// TwinCAT 3 PLC project Lynus_HTTP_Functions
// Title: Lynus HTTP Functions
// Company: Lynus AG
// ProjectVersion: 1.0.0.0
// ProgramVersion: 3.1.4023.0
// libraries:
//   Lynus Standards, * (Lynus AG)
//   Tc2_Standard, * (Beckhoff Automation GmbH)
//   Tc2_System, * (Beckhoff Automation GmbH)
//   Tc2_Utilities, * (Beckhoff Automation GmbH)
//   Tc3_IotBase, * (Beckhoff Automation GmbH)
//   Tc3_JsonXml, * (Beckhoff Automation GmbH)
//   Tc3_Module, * (Beckhoff Automation GmbH)
// project tree:
//   DUTs/Auhofcenter Vienna/ ST_ListOfVariables_Auhofcenter.TcDUT
//   DUTs/SmartMe/ ST_ListOfValues_SmartMe_ElectricMeter.TcDUT
//   DUTs/Suurstoffi Zug/Energy Part/ ST_Values_Energy_Surstoffi.TcDUT
//   DUTs/Suurstoffi Zug/Iosys Part/ ST_Values_Checked_Iosys.TcDUT, ST_Values_Iosys.TcDUT
//   DUTs/Zaptec ECS/ ST_Zaptec_ECS_State.TcDUT, ST_Zaptec_Input_Charger.TcDUT, ST_Zaptec_Input_Installation.TcDUT
//   FBs/Auhofcenter Vienna/Client FBs/ FB_GetSet_Data_Auhofcenter.TcPOU
//   FBs/Auhofcenter Vienna/Helper FBs/ FB_Decode_Json_Auhofcenter.TcPOU, FB_HTTP_Get_Auhofcenter.TcPOU
//   FBs/SmartMe/Client FBs/ FB_Get_Data_SmartMeApi_ElectricMeter.TcPOU
//   FBs/SmartMe/Helper FBs/ FB_Decode_Json_SmartMe_ElectricMeter.TcPOU, FB_HTTP_GetData_Smart_me.TcPOU
//   FBs/Suurstoffi Zug/Energy Part/Client FBs/ FB_Get_Data_Energy_Surstoffi.TcPOU
//   FBs/Suurstoffi Zug/Energy Part/Helper FBs/ FB_Decode_Json_Energy.TcPOU, FB_HTTP_Get_Energy_Surstoffi.TcPOU
//   FBs/Suurstoffi Zug/Iosys Part/Client FBs/ FB_Get_Data_Iosys.TcPOU
//   FBs/Suurstoffi Zug/Iosys Part/Helper FBs/ FB_Check_List_Iosys.TcPOU, FB_Decode_Json_Iosys.TcPOU, FB_HTTP_Get_Iosys.TcPOU
//   FBs/Zaptec ECS/Client FBs/ FB_ECS_HTTP_ZaptecAccount.TcPOU
//   FBs/Zaptec ECS/Helper FBs/ FB_HTTP_Get_Zaptec_ECS_State.TcPOU, FB_HTTP_Post_Zaptec_Current.TcPOU, FB_HTTP_Post_Zaptec_ReqToken.TcPOU

// ---- DUTs/Auhofcenter Vienna/ST_ListOfVariables_Auhofcenter.TcDUT
TYPE ST_ListOfVariables_Auhofcenter :
STRUCT
	bIsString				: BOOL;
	sVariableName			: STRING(15);
	sVariableValue			: STRING(30);
END_STRUCT
END_TYPE

// ---- DUTs/SmartMe/ST_ListOfValues_SmartMe_ElectricMeter.TcDUT
TYPE ST_ListOfValues_SmartMe_ElectricMeter :
STRUCT
	sID					: STRING(50);					//ID from the Device from the Smart-me Project
	sName				: STRING(255);					//Name from the Device from the Smart-me Project
	sActivePowerUnit 	: STRING(20);					//Unit from the Active Power from the Device from the Smart-me Project
	sCounterReadingUnit	: STRING(20);					//Unit from the Counter Reading from the Device from the Smart-me Project
	sValueDate			: STRING(30);					//Date and time when the device last sent data to the Smart Me database
	bNotAllDataIncluded	: BOOL;							//Not all Data from this Structure are included in the Response from the Device from the Smart-me Project  
	bDigitalOutput1		: BOOL;							//State from the Digital Output 1 from the Device from the Smart-me Project 
	bDigitalOutput2		: BOOL;							//State from the Digital Output 2 from the Device from the Smart-me Project
	udiActiveTariff		: UDINT;						//Actual Active tariff from the Device from the Smart-me Project
	uliSerialNr			: ULINT;						//Serial Number from the Device from the Smart-me Project
	lrPowerFactor		: LREAL;						//Power Factor from the Device from the Smart-me Project			
	lrVoltageL1			: LREAL;						//Voltage L1 from the Device from the Smart-me Project	
	lrVoltageL2			: LREAL;						//Voltage L2 from the Device from the Smart-me Project
	lrVoltageL3			: LREAL;						//Voltage L3 from the Device from the Smart-me Project
	lrCurrentL1			: LREAL;						//Current L1 from the Device from the Smart-me Project
	lrCurrentL2			: LREAL;						//Current L2 from the Device from the Smart-me Project
	lrCurrentL3			: LREAL;						//Current L3 from the Device from the Smart-me Project
	lrActivePower		: LREAL;						//Active Power from the Device from the Smart-me Project
	lrActivePowerL1		: LREAL;						//Active Power L1 from the Device from the Smart-me Project
	lrActivePowerL2		: LREAL;						//Active Power L2 from the Device from the Smart-me Project
	lrActivePowerL3		: LREAL;						//Active Power L3 from the Device from the Smart-me Project
	lrCounterReading	: LREAL;						//Counter Reading Value from the Device from the Smart-me Project
	lrCounterReadingT1	: LREAL;						//Counter Reading T1 Value from the Device from the Smart-me Project
	lrCounterReadingT2	: LREAL;						//Counter Reading T2 Value from the Device from the Smart-me Project
	lrCounterReadingT3	: LREAL;						//Counter Reading T3 Value from the Device from the Smart-me Project
	lrCounterReadingT4	: LREAL;						//Counter Reading T4 Value from the Device from the Smart-me Project
	lrCounterReadingImp	: LREAL;						//Counter Reading Import Value from the Device from the Smart-me Project
	lrCounterReadingExp	: LREAL;						//Counter Reading Export Value from the Device from the Smart-me Project
END_STRUCT
END_TYPE

// ---- DUTs/Suurstoffi Zug/Energy Part/ST_Values_Energy_Surstoffi.TcDUT
TYPE ST_Values_Energy_Surstoffi :
STRUCT
	sTimestamp			: STRING(255);						//Timestamp
	sID					: STRING(255);						//Id from the Datapoint
	lrValue				: LREAL;							//Value from the Datapoint
END_STRUCT
END_TYPE

// ---- DUTs/Suurstoffi Zug/Iosys Part/ST_Values_Checked_Iosys.TcDUT
TYPE ST_Values_Checked_Iosys :
STRUCT
	sTimestamp			: STRING(255);						//Timestamp
	sId					: STRING(255);						//Id from the Datapoint
	lrValue				: LREAL;							//Value from Datapoint
END_STRUCT
END_TYPE

// ---- DUTs/Suurstoffi Zug/Iosys Part/ST_Values_Iosys.TcDUT
{attribute 'conditionalshow'}
TYPE ST_Values_Iosys :
STRUCT
	{attribute 'hide'}
	sTimestamp			: STRING(255);					//Timestamp
	{attribute 'hide'}
	sId					: STRING(255);					//Id from the Datapoint
	{attribute 'hide'}
	sValue				: STRING(255);					//Value from Datapoint
	{attribute 'hide'}
	bNoValue			: BOOL;							//Datapoint received but without value
END_STRUCT
END_TYPE

// ---- DUTs/Zaptec ECS/ST_Zaptec_ECS_State.TcDUT
TYPE ST_Zaptec_ECS_State :
STRUCT
	bIsOnline				: BOOL;			//Shows if the Charger is Online
	bIsEnabled				: BOOL;			//Shows if the Charger is Enabled	
	rAllocatedCurrent		: REAL;			//Shows the Allocated Current in A (Only adjustable if you set via the installation API)
	rMaxCurrect				: REAL;			//Max Charge Current from Charging Station in A (Only adjustable if you set via the charger API)
	rMinCurrect				: REAL;			//Min Charge Current from Charging Station in A (Only adjustable if you set via the charger API)
	rCurrentL1				: REAL;			//Current in A from L1
	rCurrentL2				: REAL;			//Current in A from L2
	rCurrentL3				: REAL;			//Current in A from L3
	rPower					: REAL;			//Power in kW
	rEnergySession			: REAL;			//Energy in kWh from the current/last session
	diOperationMode			: DINT;			//Operation Mode form the Charger
	diWarnings				: DINT;			//Warnings from the Charger
	sChargerID				: STRING(50);	//Charger ID from Response
END_STRUCT
END_TYPE

// ---- DUTs/Zaptec ECS/ST_Zaptec_Input_Charger.TcDUT
TYPE ST_Zaptec_Input_Charger :
STRUCT
	rMinCurrentCharger					: REAL;													//Min Current for Charging Station
	rMaxCurrentCharger					: REAL;													//Max Current for Charging Station 
	sChargerID							: STRING(50);											//Charger ID
END_STRUCT
END_TYPE

// ---- DUTs/Zaptec ECS/ST_Zaptec_Input_Installation.TcDUT
TYPE ST_Zaptec_Input_Installation :
STRUCT
	rAvailableCurrentInstallation		: REAL;													//Available Current for Installation
	sInstallationID						: STRING(50);											//Installation ID
END_STRUCT
END_TYPE

// ---- FBs/Auhofcenter Vienna/Client FBs/FB_GetSet_Data_Auhofcenter.TcPOU
{attribute 'hide_all_locals'}
FUNCTION_BLOCK FB_GetSet_Data_Auhofcenter
VAR_INPUT
	bStart						: BOOL;															//Start the connection to the Service
	bWriteRequest				: BOOL;															//Send a Write Request to the Server
	bReadRequest				: BOOL;															//Send a Read Request to the Server
	tDelayRequest				: TIME := T#15S;												//Timer for delay before start with the next read or write Request
	sHostname					: STRING(255);													//Hostname or IP Adress from the Server
	arrListOfVariables			: ARRAY[1..100] OF ST_ListOfVariables_Auhofcenter;				//List of Variables what the function must be send or write		
END_VAR
VAR_OUTPUT
	bValidResult				: BOOL;															//Valid Result received from Server
    bBusy						: BOOL;															//Function is Busy
    bError						: BOOL;															//Error sucess
	bDone						: BOOL;															//True after the decoding from the received Json File
	bConnected					: BOOL;															//Connection to the Server
	arrListOfVariabelsOut		: ARRAY[1..100] OF ST_ListOfVariables_Auhofcenter;				//Received Values form the Server after read or write command
	hrErrorCode       			: HRESULT;														//Error Result from Http Client
END_VAR
VAR
	fbHttpClientEnergyHttp		: FB_IotHttpClient;												//Http Client Function
	fbHttpGet					: FB_HTTP_Get_Auhofcenter;										//Http Get Request to the Server
	fbDecodeJson				: FB_Decode_Json_Auhofcenter;									//Function to decode the received Json File
	timStartRequest				: TON;															//Timer to Start the Request
	timDissableFunctions		: TON;															//Timer to dissable the Function after Lynus_Standards.Constants_General.tTimeDissableLynusFunctions Days without connection to the Lynus Cloud
	timResetConnectionOnGVL		: TON;															//Timer to try reset the connection Flag on the GVL. (When somebody delete the Connection Function and make only a onlinechange)
	timReset24					: TON;															//timer disconnect every 24h
	FPStartRequest				: R_TRIG;														//Internal positive Edge
	FPDone						: R_TRIG;														//Internal positive Edge
	FNStart						: F_TRIG;														//Internal negative Edge
	arrListOfVariablesInt		: ARRAY[1..100] OF ST_ListOfVariables_Auhofcenter;				//Internal List of Variables to compare it with received values after a write Request	
	bErrorCheckValues			: BOOL;															//Error flag to check the values after a write Request
	byLoopCheckValues			: BYTE;															//Loop to check teh values after a Write Request. Server sends the same values back when he has received succesfully
END_VAR

//Creator : Kai Ebensperger
//Company : Lynus AG
//Date : 18.02.2021
//Version : 1.0.0.0

//With this Function is possible to send a HTTP Get Request to the System in the Auhofcenter Vienna
//Its possible to send a Send Request. Here the Server deliver the actual Values.
//On a Write Request we can send new Values to the Server.

(*-------------------------------------------------------------Service from Backend is ready and check the connection to backen for dissabel/enable Function---------------------------------------------------------------*)

//Try to reset the variable for connection on the GVL. When all is normal then the Lynus Mqtt connection function set this variable to true in the next cycle
//When we have no connection to the backend then after Lynus_Standards.Constants_General.tTimeDissableLynusFunctions days the Function is dissabled with all of his functionalities
timResetConnectionOnGVL(IN:= NOT timResetConnectionOnGVL.Q, PT:= T#1H, Q=> , ET=> );
	IF timResetConnectionOnGVL.Q THEN Lynus_Standards.GVL_Communicator.bStateConnectionToEnableFunctions := FALSE; END_IF
		IF NOT Lynus_Standards.GVL_Communicator.bStateConnectionToEnableFunctions THEN timDissableFunctions.IN := TRUE; ELSE timDissableFunctions.IN := FALSE; END_IF  
			timDissableFunctions(IN:= , PT:= Lynus_Standards.Constants_General.tTimeDissableLynusFunctions, Q=> , ET=> );

(*------------------------------------------------------------------------------------Configure HTTP Client------------------------------------------------------------------------------------------------------*)

fbHttpClientEnergyHttp.sHostName := sHostname;
fbHttpClientEnergyHttp.tConnectionTimeout := tDelayRequest;

IF NOT fbHttpClientEnergyHttp.bConfigured THEN 
	fbHttpClientEnergyHttp.nHostPort:= 80;
	fbHttpClientEnergyHttp.stTLS.bNoServerCertCheck:= FALSE;
	fbHttpClientEnergyHttp.bKeepAlive := TRUE;
	fbHttpClientEnergyHttp.tConnectionTimeout := T#10S;
END_IF

//Timer Disconnect to Server every 24H because somthing goes wrog with the loval http plc in the auhofcenter 
timReset24(IN:= bStart AND NOT timReset24.Q, PT:= T#24H, Q=> , ET=> );		

//Timer to start the Request
FPStartRequest(CLK:= bStart, Q=> );
	timStartRequest(IN:= fbHttpClientEnergyHttp.bConfigured AND bStart AND NOT timStartRequest.Q AND NOT timDissableFunctions.Q AND NOT timReset24.Q, PT:= tDelayRequest, Q=> , ET=> );
		IF ((timStartRequest.Q AND NOT bBusy) OR (FPStartRequest.Q AND NOT bBusy AND fbHttpClientEnergyHttp.bConfigured)) THEN fbHttpGet.bSend := TRUE; END_IF

IF timReset24.Q THEN fbHttpGet.bSend := FALSE; END_IF			
		
//Http Get Function
fbHttpGet(
	bWriteRequest:= bWriteRequest, 
	bReadRequest:= bReadRequest, 
	arrListOfVariables:= arrListOfVariables, 
	bSend:= , 
	tTimeOut:= T#20S,
	fbClient:= fbHttpClientEnergyHttp, 
	bValidResult=> bValidResult, 
	bBusy=> bBusy, 
	bError=> ,
	byTypeOfLastRequest=> , 
	sContent=> );

//Copy the values form the actual Request in a internal Array to compare it with the received Values when the request was a Write Request
IF fbHttpGet.bSend THEN arrListOfVariablesInt := arrListOfVariables; END_IF  
	
fbHttpGet.bSend := FALSE;
	
fbDecodeJson(
	bExecute:= fbHttpGet.bValidResult, 
	sContent:= fbHttpGet.sContent, 
	arrListOfVariabels=> arrListOfVariabelsOut, 
	bDone=> bDone, 
	bError=> );

FPDone(CLK:= bDone, Q=> );	
	
//Check after a write command if the Server has received the Values
IF fbHttpGet.byTypeOfLastRequest = 1 AND FPDone.Q THEN
	bErrorCheckValues := FALSE;
		FOR byLoopCheckValues := 1 TO 100 BY 1 DO
			IF arrListOfVariablesInt[byLoopCheckValues].sVariableName <> arrListOfVariabelsOut[byLoopCheckValues].sVariableName OR
				arrListOfVariablesInt[byLoopCheckValues].sVariableValue <> arrListOfVariabelsOut[byLoopCheckValues].sVariableValue THEN
					bErrorCheckValues := TRUE;
			END_IF	 	
		END_FOR 	
END_IF  
	
//Http Client
FNStart(CLK:= bStart, Q=> );
	IF FNStart.Q OR timReset24.Q THEN fbHttpClientEnergyHttp.Disconnect(); END_IF

fbHttpClientEnergyHttp.Execute();

//Connected
bConnected := fbHttpClientEnergyHttp.bConnected;

//Error
IF fbHttpGet.bError OR fbDecodeJson.bError OR fbHttpClientEnergyHttp.bError OR bErrorCheckValues THEN bError := TRUE; ELSE bError := FALSE; END_IF	
	hrErrorCode := fbHttpClientEnergyHttp.hrErrorCode;

END_FUNCTION_BLOCK

// ---- FBs/Auhofcenter Vienna/Helper FBs/FB_HTTP_Get_Auhofcenter.TcPOU
{attribute 'hide_all_locals'}
{attribute 'conditionalshow'}
FUNCTION_BLOCK FB_HTTP_Get_Auhofcenter
VAR_INPUT
	{attribute 'hide'}
	bWriteRequest				: BOOL;													//Send a Write Request to the Server
	{attribute 'hide'}
	bReadRequest				: BOOL;													//Send a Read Request to the Server
	{attribute 'hide'}
	arrListOfVariables			: ARRAY[1..100] OF ST_ListOfVariables_Auhofcenter;		//List of Variables what the function must be send or write
	{attribute 'hide'}
	bSend           			: BOOL;													//Send the Request
	{attribute 'hide'}
	tTimeOut					: TIME := T#10S;										//Timer for Timeout
END_VAR
VAR_IN_OUT
	{attribute 'hide'}
    fbClient          			: FB_IotHttpClient;										//HTTP Client Data
END_VAR
VAR_OUTPUT
	{attribute 'hide'}
	bValidResult				: BOOL;													//Valid Result received from Server
	{attribute 'hide'}
    bBusy             			: BOOL;													//Function is Busy
	{attribute 'hide'}
    bError           			: BOOL;													//Error sucess
	{attribute 'hide'}
	byTypeOfLastRequest			: BYTE;													//Type of the last Request. (0 = Read, 1 = Write)
	{attribute 'hide'}
	sContent         			: STRING(7500);											//Received Content
END_VAR
VAR
    fbRequest        		 	: FB_IotHttpRequest;									//Http Function
	RisingEdge        			: R_TRIG;												//Internal positive edge
	timTimeout					: TON;													//Timer for Timeout
   	bGetContentResult 			: BOOL;													//Get Content Result
	byQuantity					: BYTE;													//Quantity of Datapoints
	byLoop						: BYTE;													//Variable foor Loop to prepear the URI
	nState						: UDINT;												//Statemaschine
  	nReqCount					: UDINT;												//Counter requests
    nResCount					: UDINT;												//Counter results
    nValidResCount				: UDINT;												//Counter valid results
    nErrCount					: UDINT;												//Error Counter
	eErrorCode					: ETcIotHttpRequestError;								//Error Code
	sUriStart					: STRING(20);											//Start URI
	sUriComplete				: STRING(2000);											//Complete URI
END_VAR

//Creator : Kai Ebensperger
//Company : Lynus AG
//Date : 15.07.2021
//Version : 1.0.0.0

//With this Function is possible to send a HTTP Get Request to the System in the Auhof Center in Vienna.

//Timer for Timeout
timTimeout(IN:= nState = 1 AND bBusy, PT:= tTimeOut, Q=> , ET=> );
	IF timTimeout.Q THEN nState := 0; bBusy := FALSE; END_IF

RisingEdge(CLK:= bSend);

CASE nState OF
0:
    IF RisingEdge.Q THEN
		
		byQuantity := 0;
			FOR byLoop := 1 TO 100 BY 1 DO
				IF arrListOfVariables[byLoop].sVariableName <> '' THEN byQuantity := byQuantity + 1; END_IF 
			END_FOR
	
		sUriComplete := '';
			//Read Request
			IF bReadRequest THEN 
				sUriStart := '/lynus/read?';
					sUriComplete := sUriStart;
						IF byQuantity <= 100 THEN
							FOR byLoop := 1 TO byQuantity BY 1 DO
								CONCAT2(ADR(sUriComplete),ADR(arrListOfVariables[byLoop].sVariableName),ADR(sUriComplete),SIZEOF(sUriComplete));
									IF byLoop <= (byQuantity - 1) THEN CONCAT2(ADR(sUriComplete),ADR(','),ADR(sUriComplete),SIZEOF(sUriComplete)); END_IF	
							END_FOR
						END_IF
							byTypeOfLastRequest := 0;
			END_IF
				//Write Request
				IF bWriteRequest THEN 
					sUriStart := '/lynus/write?';
						sUriComplete := sUriStart;
							IF byQuantity <= 100 THEN
								FOR byLoop := 1 TO byQuantity BY 1 DO
									CONCAT2(ADR(sUriComplete),ADR(arrListOfVariables[byLoop].sVariableName),ADR(sUriComplete),SIZEOF(sUriComplete));
										CONCAT2(ADR(sUriComplete),ADR('='),ADR(sUriComplete),SIZEOF(sUriComplete));
											IF arrListOfVariables[byLoop].bIsString THEN CONCAT2(ADR(sUriComplete),ADR('"'),ADR(sUriComplete),SIZEOF(sUriComplete)); END_IF 	
												CONCAT2(ADR(sUriComplete),ADR(arrListOfVariables[byLoop].sVariableValue),ADR(sUriComplete),SIZEOF(sUriComplete));
													IF arrListOfVariables[byLoop].bIsString THEN CONCAT2(ADR(sUriComplete),ADR('"'),ADR(sUriComplete),SIZEOF(sUriComplete)); END_IF 			
														IF byLoop <= (byQuantity - 1) THEN CONCAT2(ADR(sUriComplete),ADR(','),ADR(sUriComplete),SIZEOF(sUriComplete)); END_IF	
								END_FOR
							END_IF
								byTypeOfLastRequest := 1;	
				END_IF
		
		bValidResult := FALSE;
		
		IF fbRequest.SendRequest(sUri:= sUriComplete,
								 fbClient:= fbClient, 
									eRequestType:= ETcIotHttpRequestType.HTTP_Get, 0, 0, 0) THEN
			nState:= 1;
			nReqCount:= nReqCount+1;
			bBusy:= TRUE;
			bError:= FALSE;
		END_IF
    END_IF
	
1:
    IF NOT fbRequest.bBusy THEN
       IF NOT fbRequest.bError THEN
            bGetContentResult:= fbRequest.GetContent(pContent:= ADR(sContent), 
                                                     nContentSize:= SIZEOF(sContent), 
                                                     bSetNullTermination:= TRUE);
            IF fbRequest.nStatusCode >= 200 AND fbRequest.nStatusCode < 300 THEN
                	bValidResult := TRUE;
                    nValidResCount:= nValidResCount+1;
                    bError:= FALSE;
               		nResCount:= nResCount+1;
           END_IF
		   		//Error Response from the Server
				IF sContent = 'Error' THEN bError := TRUE; END_IF
        END_IF
			IF fbRequest.bError THEN bError:= TRUE; eErrorCode := fbRequest.eErrorId; END_IF 
			nState:= 0;
			bBusy:= FALSE;
			IF bError THEN
				nErrCount:= nErrCount+1;
			END_IF	
    END_IF
	
END_CASE

END_FUNCTION_BLOCK

// ---- FBs/Auhofcenter Vienna/Helper FBs/FB_Decode_Json_Auhofcenter.TcPOU
{attribute 'hide_all_locals'}
{attribute 'conditionalshow'}
FUNCTION_BLOCK FB_Decode_Json_Auhofcenter
VAR_INPUT
	{attribute 'hide'}
	bExecute						: BOOL;																			//Start the decoding from the Json File
	{attribute 'hide'}
	sContent         				: STRING(7500);																	//Received Content
END_VAR
VAR_OUTPUT
	{attribute 'hide'}
	arrListOfVariabels				: ARRAY[1..100] OF ST_ListOfVariables_Auhofcenter;								//List with all received Values from the Server
	{attribute 'hide'}
	bDone							: BOOL;																			//True when the decoding is done
	{attribute 'hide'}
	bError							: BOOL;																			//Error Bit
END_VAR
VAR
	fbJsonRead					    : FB_JsonDomParser;																//FB Json Dom reader
 	jsonDocInit  					: SJsonValue;																	//Json value
	jsonDoc		  					: SJsonValue;																	//Json value
	jsonPropID   					: SJsonValue;																	//Json value
	jsonIteratorArrayStart			: SJsonAIterator;																//Json AIterator
	jsonIteratorArrayEnd			: SJsonAIterator;																//Json AIterator
	FPExecute						: R_TRIG;																		//Internal positive edge
	byCounterForArray				: BYTE;																			//Counter to fill the output array with conntent
	byLoopInit						: BYTE;																			//Loop to clear the output array before fill the new content inside
END_VAR

//Creator : Kai Ebensperger
//Company : Lynus AG
//Date : 15.07.2021
//Version : 1.0.0.0

//With this Function we can decode the received Json form the System in the Auhofcenter in Vienna

bDone := FALSE;

FPExecute(CLK:= bExecute, Q=> );

//Start with the Json Doc
jsonDocInit := fbJsonRead.ParseDocument(sContent);

IF FPExecute.Q THEN
	byCounterForArray := 0;	
		bError := FALSE;

	//Clear the Output for new Values
	FOR byLoopInit := 1 TO 100 BY 1 DO
		arrListOfVariabels[byLoopInit].bIsString := FALSE;
			arrListOfVariabels[byLoopInit].sVariableName := '';
				arrListOfVariabels[byLoopInit].sVariableValue := '';
	END_FOR
	
	//Check if the values are inside of a Array 		
	IF jsonDocInit <> 0 THEN
		IF fbJsonRead.IsArray(jsonDocInit) THEN
			jsonIteratorArrayStart := fbJsonRead.ArrayBegin(jsonDocInit);	
				jsonIteratorArrayEnd := fbJsonRead.ArrayEnd(jsonDocInit);
		ELSE
			bError := TRUE;
		END_IF
	ELSE
		bError := TRUE;
	END_IF
		//Start to Decode the Json File
		IF jsonDocInit <> 0 AND jsonIteratorArrayStart <> 0 AND jsonIteratorArrayEnd <> 0 AND NOT bError THEN
		
			WHILE jsonIteratorArrayStart <> jsonIteratorArrayEnd DO  
				jsonDoc := fbJsonRead.GetArrayValue(jsonIteratorArrayStart);
					//Find the Member ID
					jsonPropID := fbJsonRead.FindMember(jsonDoc, 'ID');	
						IF jsonPropID <> 0 THEN
							IF fbJsonRead.IsString(jsonPropID) THEN
								byCounterForArray := byCounterForArray + 1;
									byCounterForArray := LIMIT(1,byCounterForArray,100);	
										arrListOfVariabels[byCounterForArray].sVariableName := fbJsonRead.GetString(jsonPropID);
							ELSE
								bError := TRUE;	
							END_IF	
						END_IF 
					//Find the Member v
					jsonPropID := fbJsonRead.FindMember(jsonDoc, 'v');
						IF jsonPropID <> 0 THEN
							IF fbJsonRead.IsNumber(jsonPropID) THEN
								arrListOfVariabels[byCounterForArray].sVariableValue := LREAL_TO_STRING(fbJsonRead.GetDouble(jsonPropID));
							ELSE
								bError := TRUE;		
							END_IF
						END_IF
					//Find the Member vs
					jsonPropID := fbJsonRead.FindMember(jsonDoc, 'vs');
						IF jsonPropID <> 0 THEN
							IF fbJsonRead.IsString(jsonPropID) THEN
								arrListOfVariabels[byCounterForArray].sVariableValue := fbJsonRead.GetString(jsonPropID);
									arrListOfVariabels[byCounterForArray].bIsString := TRUE;
							ELSE
								bError := TRUE;	
							END_IF
						END_IF
					jsonIteratorArrayStart := fbJsonRead.NextArray(jsonIteratorArrayStart);
			END_WHILE
				bDone := TRUE;
		END_IF
END_IF

END_FUNCTION_BLOCK

// ---- FBs/SmartMe/Client FBs/FB_Get_Data_SmartMeApi_ElectricMeter.TcPOU
{attribute 'hide_all_locals'}
FUNCTION_BLOCK FB_Get_Data_SmartMeApi_ElectricMeter
VAR_INPUT
	bStart						: BOOL;															//Start the connection to the Service
	sUsername					: STRING(50);													//Username from the smart-me Project
	sPassword					: STRING(50);													//Password from the smart-me Project
	tDelayRequest				: TIME := T#1S; 												//Delay between the Requests		
END_VAR
VAR_OUTPUT
	bValidResult				: BOOL;															//Valid Result received from Server
    bBusy						: BOOL;															//Function is Busy
    bError						: BOOL;															//Error sucess
	hrErrorCode       			: HRESULT;														//Error Result from Http Client
	arrListOfDevices			: ARRAY[1..50] OF ST_ListOfValues_SmartMe_ElectricMeter;		//List with all received Values from the Server
END_VAR
VAR
	fbHttpClientSmartMe			: FB_IotHttpClient :=(sHostName:='smart-me.com',
                                  bKeepAlive:=TRUE, tConnectionTimeout:=T#15S);					//Http Client Function
	fbHttpGet					: FB_HTTP_GetData_Smart_me;										//Http Get Request to the Smart Me Service
	fbJson						: FB_Decode_Json_SmartMe_ElectricMeter;							//Deconde received Json
	timStartRequest				: TON;															//Timer to Start the Request
	timDissableFunctions		: TON;															//Timer to dissable the Function after Lynus_Standards.Constants_General.tTimeDissableLynusFunctions Days without connection to the Lynus Cloud
	timResetConnectionOnGVL		: TON;															//Timer to try reset the connection Flag on the GVL. (When somebody delete the Connection Function and make only a onlinechange)
	timReset24					: TON;															//timer disconnect every 24h
	FPStartRequest				: R_TRIG;														//Internal positive Edge
	FNStart						: F_TRIG;														//Internal negative Edge
END_VAR

//Creator : Kai Ebensperger
//Company : Lynus AG
//Date : 29.09.2021
//Version : 1.0.0.0

//With this Function is possible to send a HTTP Get Request to the Smart-me System and recieve values from the Project wich is defined with the Username and the password
//With this Function is possible to decode only Data from Electric Meter in the Project
//Other Device Types or Meters are not supported and the Function deliver a Error
//Attetnion : If the Username is a Mailadress write all in small carakters. For example kai.ebensperger@ventus.ag

(*--------------------------------------------------------------------------------------------------------Limits---------------------------------------------------------------------------------------------------*)

tDelayRequest := LIMIT(T#1S,tDelayRequest,T#15M);

(*-------------------------------------------------------------Service from Backend is ready and check the connection to backen for dissabel/enable Function---------------------------------------------------------------*)

//Try to reset the variable for connection on the GVL. When all is normal then the Lynus Mqtt connection function set this variable to true in the next cycle
//When we have no connection to the backend then after Lynus_Standards.Constants_General.tTimeDissableLynusFunctions days the Function is dissabled with all of his functionalities
timResetConnectionOnGVL(IN:= NOT timResetConnectionOnGVL.Q, PT:= T#1H, Q=> , ET=> );
	IF timResetConnectionOnGVL.Q THEN Lynus_Standards.GVL_Communicator.bStateConnectionToEnableFunctions := FALSE; END_IF
		IF NOT Lynus_Standards.GVL_Communicator.bStateConnectionToEnableFunctions THEN timDissableFunctions.IN := TRUE; ELSE timDissableFunctions.IN := FALSE; END_IF  
			timDissableFunctions(IN:= , PT:= Lynus_Standards.Constants_General.tTimeDissableLynusFunctions, Q=> , ET=> );

(*------------------------------------------------------------------------------------Configure HTTP Client------------------------------------------------------------------------------------------------------*)

IF NOT fbHttpClientSmartMe.bConfigured THEN
    fbHttpClientSmartMe.nHostPort:= 443;
    fbHttpClientSmartMe.stTLS.bNoServerCertCheck:= TRUE;
END_IF

//Timer Disconnect to Server every 24H because somthing goes wrog with the loval http plc in the auhofcenter 
timReset24(IN:= bStart AND NOT timReset24.Q, PT:= T#24H, Q=> , ET=> );

//Timer to start the Request
FPStartRequest(CLK:= bStart, Q=> );
	timStartRequest(IN:= bStart AND NOT timStartRequest.Q AND NOT timDissableFunctions.Q AND NOT bBusy AND fbHttpClientSmartMe.bConfigured AND NOT timReset24.Q, PT:= tDelayRequest, Q=> , ET=> );
		IF timStartRequest.Q OR (FPStartRequest.Q AND NOT bBusy AND fbHttpClientSmartMe.bConfigured) THEN fbHttpGet.bSend := TRUE; END_IF

IF timReset24.Q THEN fbHttpGet.bSend := FALSE; END_IF				
		
//Http Get Function
fbHttpGet(
	bSend:= , 
	sUsername:= sUsername, 
	sPassword:= sPassword, 
	tTimeOut:= T#20S,
	fbClient:= fbHttpClientSmartMe, 
	bValidResult=> bValidResult, 
	bBusy=> bBusy, 
	bError=> , 
	sContent=> );
	
fbHttpGet.bSend := FALSE;
	
//Decode Json
fbJson(
	bExecute:= bValidResult, 
	sContent:= fbHttpGet.sContent, 
	arrListOfDevices=> , 
	bDone=> , 
	bError=> );

IF fbJson.bDone AND NOT fbJson.bError AND NOT bBusy THEN
	arrListOfDevices := fbJson.arrListOfDevices;
END_IF		
	
//Http Client
FNStart(CLK:= bStart, Q=> );
	IF FNStart.Q OR timReset24.Q THEN fbHttpClientSmartMe.Disconnect(); END_IF

fbHttpClientSmartMe.Execute();

//Error
IF fbHttpGet.bError OR fbJson.bError OR fbHttpClientSmartMe.bError THEN bError := TRUE; ELSE bError := FALSE; END_IF	
	hrErrorCode := fbHttpClientSmartMe.hrErrorCode;

END_FUNCTION_BLOCK

// ---- FBs/SmartMe/Helper FBs/FB_HTTP_GetData_Smart_me.TcPOU
{attribute 'hide_all_locals'}
{attribute 'conditionalshow'}
FUNCTION_BLOCK FB_HTTP_GetData_Smart_me
VAR_INPUT
	{attribute 'hide'}
   	bSend               : BOOL;													//Send the Request to the Service
	{attribute 'hide'}
	sUsername			: STRING(50);											//Username from the smart-me Project
	{attribute 'hide'}
	sPassword			: STRING(50);											//Password from the smart-me Project
	{attribute 'hide'}
	tTimeOut			: TIME := T#10S;										//Timer for Timeout
END_VAR
VAR_IN_OUT
	{attribute 'hide'}
    fbClient            : FB_IotHttpClient;										//Connection to the HTTP Client Function
END_VAR
VAR_OUTPUT
	{attribute 'hide'}
	bValidResult		: BOOL;													//Valid Result received from Server
	{attribute 'hide'}
    bBusy               : BOOL;													//Function is Busy
	{attribute 'hide'}
    bError              : BOOL;													//Function has a error
	{attribute 'hide'}
	sContent            : STRING(30000);										//Received Content
END_VAR
VAR
	fbRequest           : FB_IotHttpRequest;									//Http Request Function
    fbHeader            : FB_IotHttpHeaderFieldMap;								//Header Function
	fbJsonWrite     	: FB_JsonSaxWriter;										//Json Write function to generate the based64 Part for the Header
 	timTimeout			: TON;													//Timer for Timeout
	RisingEdge          : R_TRIG;												//Internal rising edge
   	bGetContentResult   : BOOL;													//True when we receive content												
    nState              : UDINT;												//Statemachine for the http request
    nReqCount           : UDINT;												//Request Counter
    nResCount           : UDINT;												//Receive Counter
    nValidResCount      : UDINT;												//Valid Receive Counter
    nErrCount           : UDINT;												//Error Counter
    bOnce               : BOOL:= TRUE;											//Add the addidional Header Part
	sbase64				: STRING(255);											//Based 64 string from the username and Password
	sbase64_CP			: STRING(255);											//Based 64 string from the username and Password to compare it and modify the header
	sCompleteString		: STRING(101);											//Complete string with username and password
	iLen				: INT;													//Lengh from the string
END_VAR

//Creator : Kai Ebensperger
//Company : Lynus AG
//Date : 29.09.2021
//Version : 1.0.0.0

//With this Function its possible to make a Request to the smart-me Database to receive Information from a Project and his devices.

//Convert the Username and the password from string to Ascii and then in a Based64 format
sCompleteString := CONCAT(CONCAT(sUsername,':'),sPassword);
	iLen := LEN(sCompleteString); 
		fbJsonWrite.AddBase64(ADR(sCompleteString),iLen);
			sbase64 := fbJsonWrite.GetDocument();
				fbJsonWrite.ResetDocument();

sbase64 := DELETE(sbase64,1,FIND(sbase64,'"'));	
	sbase64 := DELETE(sbase64,1,FIND(sbase64,'"'));		
	
sbase64 := CONCAT('Basic ',sbase64);

//Add Username and Password to the Header of the Request
IF sbase64 <> sbase64_CP AND nState = 0 THEN bOnce := TRUE; sbase64_CP := sbase64; END_IF  

IF bOnce THEN
    fbHeader.AddField('Authorization',sbase64, FALSE);
    bOnce:= FALSE;
END_IF

//Timer for Timeout
timTimeout(IN:= nState = 1 AND bBusy, PT:= tTimeOut, Q=> , ET=> );
	IF timTimeout.Q THEN nState := 0; bBusy := FALSE; END_IF

//Statemachine to generate the Request

RisingEdge(CLK:= bSend);
	CASE nState OF
		
		0://Request
			IF RisingEdge.Q THEN
				IF fbRequest.SendRequest(sUri:= '/api/Devices', fbClient:= fbClient, 
										 eRequestType:= ETcIotHttpRequestType.HTTP_GET, 0, 0, fbHeader) THEN
					nState:= 1;
					nReqCount:= nReqCount + 1;
					bBusy:= TRUE;
					bError:= FALSE;
					bValidResult := FALSE;
				END_IF
			END_IF
			
		1://Wait for the Response
			IF NOT fbRequest.bBusy THEN
				bError:= TRUE;
					IF NOT fbRequest.bError THEN
						bGetContentResult:= fbRequest.GetContent(pContent:= ADR(sContent),
																 nContentSize:= SIZEOF(sContent), 
																 bSetNullTermination:= TRUE);
						IF fbRequest.nStatusCode >= 200 AND fbRequest.nStatusCode < 300 THEN
							bValidResult := TRUE;
							nResCount:= nResCount + 1;
							bError:= FALSE;
						END_IF
					END_IF
						nState:= 0;
						bBusy:= FALSE;
							IF bError THEN
								nErrCount:= nErrCount + 1;
							END_IF
			END_IF
			
	END_CASE

END_FUNCTION_BLOCK

// ---- FBs/SmartMe/Helper FBs/FB_Decode_Json_SmartMe_ElectricMeter.TcPOU
{attribute 'hide_all_locals'}
{attribute 'conditionalshow'}
FUNCTION_BLOCK FB_Decode_Json_SmartMe_ElectricMeter
VAR_INPUT
	{attribute 'hide'}
	bExecute						: BOOL;																			//Start the decoding from the Json File
	{attribute 'hide'}
	sContent         				: STRING(30000);																//Received Content
END_VAR
VAR_OUTPUT
	{attribute 'hide'}
	arrListOfDevices				: ARRAY[1..50] OF ST_ListOfValues_SmartMe_ElectricMeter;						//List with all received Values from the Server
	{attribute 'hide'}
	bDone							: BOOL;																			//True when the decoding is done
	{attribute 'hide'}
	bError							: BOOL;																			//Error Bit
END_VAR
VAR
	fbJsonRead					    : FB_JsonDomParser;																//FB Json Dom reader
 	jsonDocInit  					: SJsonValue;																	//Json value
	jsonDoc		  					: SJsonValue;																	//Json value
	jsonPropID   					: SJsonValue;																	//Json value
	jsonIteratorArrayStart			: SJsonAIterator;																//Json AIterator
	jsonIteratorArrayEnd			: SJsonAIterator;																//Json AIterator
	FPExecute						: R_TRIG;																		//Internal positive edge
	byCounterForArray				: BYTE;																			//Counter to fill the output array with conntent
	byLoopInit						: BYTE;																			//Loop to clear the output array before fill the new content inside
END_VAR

//Creator : Kai Ebensperger
//Company : Lynus AG
//Date : 29.09.2021
//Version : 1.0.0.0

//With this Function we can decode the received Json form a Smart-Me Project
//With this Function its possible to decode only the Data from Electric Meter from the Smart-me Project
//Other Devices are not supported with this function 

bDone := FALSE;

FPExecute(CLK:= bExecute, Q=> );

//Start with the Json Doc
jsonDocInit := fbJsonRead.ParseDocument(sContent);

IF FPExecute.Q THEN
	byCounterForArray := 0;	
		bError := FALSE;

	//Clear the Output for new Values
	FOR byLoopInit := 1 TO 50 BY 1 DO
		arrListOfDevices[byLoopInit].lrActivePower := 0;
			arrListOfDevices[byLoopInit].sActivePowerUnit := '';
				arrListOfDevices[byLoopInit].sID := '';
					arrListOfDevices[byLoopInit].sName := '';
						arrListOfDevices[byLoopInit].uliSerialNr := 0;
							arrListOfDevices[byLoopInit].sValueDate := '';	
								arrListOfDevices[byLoopInit].sCounterReadingUnit := '';
									arrListOfDevices[byLoopInit].bDigitalOutput1 := FALSE;
										arrListOfDevices[byLoopInit].bDigitalOutput2 := FALSE;
											arrListOfDevices[byLoopInit].bNotAllDataIncluded := FALSE;
												arrListOfDevices[byLoopInit].udiActiveTariff := 0;
													arrListOfDevices[byLoopInit].lrPowerFactor := 0;
														arrListOfDevices[byLoopInit].lrVoltageL1 := 0;
															arrListOfDevices[byLoopInit].lrVoltageL2 := 0;
																arrListOfDevices[byLoopInit].lrVoltageL3 := 0;
																	arrListOfDevices[byLoopInit].lrCurrentL1 := 0;
																		arrListOfDevices[byLoopInit].lrCurrentL2 := 0;
																			arrListOfDevices[byLoopInit].lrCurrentL3 := 0;
																				arrListOfDevices[byLoopInit].lrActivePowerL1 := 0;
																					arrListOfDevices[byLoopInit].lrActivePowerL2 := 0;
																						arrListOfDevices[byLoopInit].lrActivePowerL3 := 0;
																							arrListOfDevices[byLoopInit].lrCounterReading := 0;
																								arrListOfDevices[byLoopInit].lrCounterReadingT1 := 0;
																									arrListOfDevices[byLoopInit].lrCounterReadingT2 := 0;
																										arrListOfDevices[byLoopInit].lrCounterReadingT3 := 0;
																											arrListOfDevices[byLoopInit].lrCounterReadingT4 := 0;
																												arrListOfDevices[byLoopInit].lrCounterReadingImp := 0;	
																													arrListOfDevices[byLoopInit].lrCounterReadingExp := 0;
	END_FOR
	
	//Check if the values are inside of a Array 		
	IF jsonDocInit <> 0 THEN
		IF fbJsonRead.IsArray(jsonDocInit) THEN
			jsonIteratorArrayStart := fbJsonRead.ArrayBegin(jsonDocInit);	
				jsonIteratorArrayEnd := fbJsonRead.ArrayEnd(jsonDocInit);
		ELSE
			bError := TRUE;
		END_IF
	ELSE
		bError := TRUE;
	END_IF
		//Start to Decode the Json File
		IF jsonDocInit <> 0 AND jsonIteratorArrayStart <> 0 AND jsonIteratorArrayEnd <> 0 AND NOT bError THEN
		
			WHILE jsonIteratorArrayStart <> jsonIteratorArrayEnd DO  
				jsonDoc := fbJsonRead.GetArrayValue(jsonIteratorArrayStart);
(*--------------------------------------------------------------------------------------------------Must have Members--------------------------------------------------------------------------------------------------------*)
					//Find the Member Id
					jsonPropID := fbJsonRead.FindMember(jsonDoc, 'Id');	
						IF jsonPropID <> 0 THEN
							IF fbJsonRead.IsString(jsonPropID) THEN
								byCounterForArray := byCounterForArray + 1;
									byCounterForArray := LIMIT(1,byCounterForArray,50);	
										arrListOfDevices[byCounterForArray].sID := fbJsonRead.GetString(jsonPropID);
							ELSE
								bError := TRUE;	
							END_IF	
						END_IF 
					//Find the Member Name
					jsonPropID := fbJsonRead.FindMember(jsonDoc, 'Name');
						IF jsonPropID <> 0 THEN
							IF fbJsonRead.IsString(jsonPropID) THEN
								arrListOfDevices[byCounterForArray].sName := fbJsonRead.GetString(jsonPropID);
							ELSE
								bError := TRUE;		
							END_IF
						END_IF
					//Find the Member Serial
					jsonPropID := fbJsonRead.FindMember(jsonDoc, 'Serial');
						IF jsonPropID <> 0 THEN
							IF fbJsonRead.IsUint64(jsonPropID) THEN
								arrListOfDevices[byCounterForArray].uliSerialNr := fbJsonRead.GetUint64(jsonPropID);
							ELSE
								bError := TRUE;	
							END_IF
						END_IF
					//Find the Member Active Power
					jsonPropID := fbJsonRead.FindMember(jsonDoc, 'ActivePower');
						IF jsonPropID <> 0 THEN
							IF fbJsonRead.IsNumber(jsonPropID) THEN
								arrListOfDevices[byCounterForArray].lrActivePower := fbJsonRead.GetDouble(jsonPropID);
									//Limit for 2 commas
									IF arrListOfDevices[byCounterForArray].lrActivePower >= - 999999999999999 AND arrListOfDevices[byCounterForArray].lrActivePower <= 999999999999999 THEN
										arrListOfDevices[byCounterForArray].lrActivePower := LINT_TO_LREAL(LREAL_TO_LINT((arrListOfDevices[byCounterForArray].lrActivePower) * 100)) / 100;	
									END_IF 
							ELSE
								bError := TRUE;		
							END_IF
						END_IF
					//Find the Member Active Power Unit
					jsonPropID := fbJsonRead.FindMember(jsonDoc, 'ActivePowerUnit');
						IF jsonPropID <> 0 THEN
							IF fbJsonRead.IsString(jsonPropID) THEN
								arrListOfDevices[byCounterForArray].sActivePowerUnit := fbJsonRead.GetString(jsonPropID);
							ELSE
								bError := TRUE;		
							END_IF
						END_IF
					//Find the Member Value Date
					jsonPropID := fbJsonRead.FindMember(jsonDoc, 'ValueDate');
						IF jsonPropID <> 0 THEN
							IF fbJsonRead.IsString(jsonPropID) THEN
								arrListOfDevices[byCounterForArray].sValueDate := fbJsonRead.GetString(jsonPropID);
							ELSE
								bError := TRUE;		
							END_IF
						END_IF
(*--------------------------------------------------------------------------------------------------Additional Members--------------------------------------------------------------------------------------------------------*)
					//Find the Member Counter Reading Unit
					jsonPropID := fbJsonRead.FindMember(jsonDoc, 'CounterReadingUnit');
						IF jsonPropID <> 0 THEN
							IF fbJsonRead.IsString(jsonPropID) THEN
								arrListOfDevices[byCounterForArray].sCounterReadingUnit := fbJsonRead.GetString(jsonPropID);
							END_IF
						ELSE
							arrListOfDevices[byCounterForArray].bNotAllDataIncluded := TRUE;
						END_IF
					//Find the Member Digital Output 1
					jsonPropID := fbJsonRead.FindMember(jsonDoc, 'DigitalOutput1');
						IF jsonPropID <> 0 THEN
							IF fbJsonRead.IsBool(jsonPropID) THEN
								arrListOfDevices[byCounterForArray].bDigitalOutput1 := fbJsonRead.GetBool(jsonPropID);
							END_IF
						ELSE
							arrListOfDevices[byCounterForArray].bNotAllDataIncluded := TRUE;
						END_IF
					//Find the Member Digital Output 2
					jsonPropID := fbJsonRead.FindMember(jsonDoc, 'DigitalOutput2');
						IF jsonPropID <> 0 THEN
							IF fbJsonRead.IsBool(jsonPropID) THEN
								arrListOfDevices[byCounterForArray].bDigitalOutput2 := fbJsonRead.GetBool(jsonPropID);
							END_IF
						ELSE
							arrListOfDevices[byCounterForArray].bNotAllDataIncluded := TRUE;
						END_IF
					//Find the Member ActiveTariff
					jsonPropID := fbJsonRead.FindMember(jsonDoc, 'ActiveTariff');
						IF jsonPropID <> 0 THEN
							IF fbJsonRead.IsUint(jsonPropID) THEN
								arrListOfDevices[byCounterForArray].udiActiveTariff := fbJsonRead.GetUint(jsonPropID);
							END_IF
						ELSE
							arrListOfDevices[byCounterForArray].bNotAllDataIncluded := TRUE;
						END_IF
					//Find the Member PowerFactor
					jsonPropID := fbJsonRead.FindMember(jsonDoc, 'PowerFactor');
						IF jsonPropID <> 0 THEN
							IF fbJsonRead.IsNumber(jsonPropID) THEN
								arrListOfDevices[byCounterForArray].lrPowerFactor := fbJsonRead.GetDouble(jsonPropID);
									//Limit for 2 commas
									IF arrListOfDevices[byCounterForArray].lrPowerFactor >= - 999999999999999 AND arrListOfDevices[byCounterForArray].lrPowerFactor <= 999999999999999 THEN
										arrListOfDevices[byCounterForArray].lrPowerFactor := LINT_TO_LREAL(LREAL_TO_LINT((arrListOfDevices[byCounterForArray].lrPowerFactor) * 100)) / 100;	
									END_IF	
							END_IF
						ELSE
							arrListOfDevices[byCounterForArray].bNotAllDataIncluded := TRUE;
						END_IF
					//Find the Member Voltage L1
					jsonPropID := fbJsonRead.FindMember(jsonDoc, 'VoltageL1');
						IF jsonPropID <> 0 THEN
							IF fbJsonRead.IsNumber(jsonPropID) THEN
								arrListOfDevices[byCounterForArray].lrVoltageL1 := fbJsonRead.GetDouble(jsonPropID);
									//Limit for 2 commas
									IF arrListOfDevices[byCounterForArray].lrVoltageL1 >= - 999999999999999 AND arrListOfDevices[byCounterForArray].lrVoltageL1 <= 999999999999999 THEN
										arrListOfDevices[byCounterForArray].lrVoltageL1 := LINT_TO_LREAL(LREAL_TO_LINT((arrListOfDevices[byCounterForArray].lrVoltageL1) * 100)) / 100;	
									END_IF	
							END_IF
						ELSE
							arrListOfDevices[byCounterForArray].bNotAllDataIncluded := TRUE;
						END_IF
					//Find the Member Voltage L2
					jsonPropID := fbJsonRead.FindMember(jsonDoc, 'VoltageL2');
						IF jsonPropID <> 0 THEN
							IF fbJsonRead.IsNumber(jsonPropID) THEN
								arrListOfDevices[byCounterForArray].lrVoltageL2 := fbJsonRead.GetDouble(jsonPropID);
									//Limit for 2 commas
									IF arrListOfDevices[byCounterForArray].lrVoltageL2 >= - 999999999999999 AND arrListOfDevices[byCounterForArray].lrVoltageL2 <= 999999999999999 THEN
										arrListOfDevices[byCounterForArray].lrVoltageL2 := LINT_TO_LREAL(LREAL_TO_LINT((arrListOfDevices[byCounterForArray].lrVoltageL2) * 100)) / 100;	
									END_IF	
							END_IF
						ELSE
							arrListOfDevices[byCounterForArray].bNotAllDataIncluded := TRUE;
						END_IF
					//Find the Member Voltage L3
					jsonPropID := fbJsonRead.FindMember(jsonDoc, 'VoltageL3');
						IF jsonPropID <> 0 THEN
							IF fbJsonRead.IsNumber(jsonPropID) THEN
								arrListOfDevices[byCounterForArray].lrVoltageL3 := fbJsonRead.GetDouble(jsonPropID);
									//Limit for 2 commas
									IF arrListOfDevices[byCounterForArray].lrVoltageL3 >= - 999999999999999 AND arrListOfDevices[byCounterForArray].lrVoltageL3 <= 999999999999999 THEN
										arrListOfDevices[byCounterForArray].lrVoltageL3 := LINT_TO_LREAL(LREAL_TO_LINT((arrListOfDevices[byCounterForArray].lrVoltageL3) * 100)) / 100;	
									END_IF	
							END_IF
						ELSE
							arrListOfDevices[byCounterForArray].bNotAllDataIncluded := TRUE;
						END_IF
					//Find the Member Current L1
					jsonPropID := fbJsonRead.FindMember(jsonDoc, 'CurrentL1');
						IF jsonPropID <> 0 THEN
							IF fbJsonRead.IsNumber(jsonPropID) THEN
								arrListOfDevices[byCounterForArray].lrCurrentL1 := fbJsonRead.GetDouble(jsonPropID);
									//Limit for 2 commas
									IF arrListOfDevices[byCounterForArray].lrCurrentL1 >= - 999999999999999 AND arrListOfDevices[byCounterForArray].lrCurrentL1 <= 999999999999999 THEN
										arrListOfDevices[byCounterForArray].lrCurrentL1 := LINT_TO_LREAL(LREAL_TO_LINT((arrListOfDevices[byCounterForArray].lrCurrentL1) * 100)) / 100;	
									END_IF	
							END_IF
						ELSE
							arrListOfDevices[byCounterForArray].bNotAllDataIncluded := TRUE;
						END_IF
					//Find the Member Current L2
					jsonPropID := fbJsonRead.FindMember(jsonDoc, 'CurrentL2');
						IF jsonPropID <> 0 THEN
							IF fbJsonRead.IsNumber(jsonPropID) THEN
								arrListOfDevices[byCounterForArray].lrCurrentL2 := fbJsonRead.GetDouble(jsonPropID);
									//Limit for 2 commas
									IF arrListOfDevices[byCounterForArray].lrCurrentL2 >= - 999999999999999 AND arrListOfDevices[byCounterForArray].lrCurrentL2 <= 999999999999999 THEN
										arrListOfDevices[byCounterForArray].lrCurrentL2 := LINT_TO_LREAL(LREAL_TO_LINT((arrListOfDevices[byCounterForArray].lrCurrentL2) * 100)) / 100;	
									END_IF	
							END_IF
						ELSE
							arrListOfDevices[byCounterForArray].bNotAllDataIncluded := TRUE;
						END_IF
					//Find the Member Current L3
					jsonPropID := fbJsonRead.FindMember(jsonDoc, 'CurrentL3');
						IF jsonPropID <> 0 THEN
							IF fbJsonRead.IsNumber(jsonPropID) THEN
								arrListOfDevices[byCounterForArray].lrCurrentL3 := fbJsonRead.GetDouble(jsonPropID);
									//Limit for 2 commas
									IF arrListOfDevices[byCounterForArray].lrCurrentL3 >= - 999999999999999 AND arrListOfDevices[byCounterForArray].lrCurrentL3 <= 999999999999999 THEN
										arrListOfDevices[byCounterForArray].lrCurrentL3 := LINT_TO_LREAL(LREAL_TO_LINT((arrListOfDevices[byCounterForArray].lrCurrentL3) * 100)) / 100;	
									END_IF	
							END_IF
						ELSE
							arrListOfDevices[byCounterForArray].bNotAllDataIncluded := TRUE;
						END_IF
					//Find the Member Active Power L1
					jsonPropID := fbJsonRead.FindMember(jsonDoc, 'ActivePowerL1');
						IF jsonPropID <> 0 THEN
							IF fbJsonRead.IsNumber(jsonPropID) THEN
								arrListOfDevices[byCounterForArray].lrActivePowerL1 := fbJsonRead.GetDouble(jsonPropID);
									//Limit for 2 commas
									IF arrListOfDevices[byCounterForArray].lrActivePowerL1 >= - 999999999999999 AND arrListOfDevices[byCounterForArray].lrActivePowerL1 <= 999999999999999 THEN
										arrListOfDevices[byCounterForArray].lrActivePowerL1 := LINT_TO_LREAL(LREAL_TO_LINT((arrListOfDevices[byCounterForArray].lrActivePowerL1) * 100)) / 100;	
									END_IF	
							END_IF
						ELSE
							arrListOfDevices[byCounterForArray].bNotAllDataIncluded := TRUE;
						END_IF
					//Find the Member Active Power L2
					jsonPropID := fbJsonRead.FindMember(jsonDoc, 'ActivePowerL2');
						IF jsonPropID <> 0 THEN
							IF fbJsonRead.IsNumber(jsonPropID) THEN
								arrListOfDevices[byCounterForArray].lrActivePowerL2 := fbJsonRead.GetDouble(jsonPropID);
									//Limit for 2 commas
									IF arrListOfDevices[byCounterForArray].lrActivePowerL2 >= - 999999999999999 AND arrListOfDevices[byCounterForArray].lrActivePowerL2 <= 999999999999999 THEN
										arrListOfDevices[byCounterForArray].lrActivePowerL2 := LINT_TO_LREAL(LREAL_TO_LINT((arrListOfDevices[byCounterForArray].lrActivePowerL2) * 100)) / 100;	
									END_IF	
							END_IF
						ELSE
							arrListOfDevices[byCounterForArray].bNotAllDataIncluded := TRUE;
						END_IF
					//Find the Member Active Power L3
					jsonPropID := fbJsonRead.FindMember(jsonDoc, 'ActivePowerL3');
						IF jsonPropID <> 0 THEN
							IF fbJsonRead.IsNumber(jsonPropID) THEN
								arrListOfDevices[byCounterForArray].lrActivePowerL3 := fbJsonRead.GetDouble(jsonPropID);
									//Limit for 2 commas
									IF arrListOfDevices[byCounterForArray].lrActivePowerL3 >= - 999999999999999 AND arrListOfDevices[byCounterForArray].lrActivePowerL3 <= 999999999999999 THEN
										arrListOfDevices[byCounterForArray].lrActivePowerL3 := LINT_TO_LREAL(LREAL_TO_LINT((arrListOfDevices[byCounterForArray].lrActivePowerL3) * 100)) / 100;	
									END_IF	
							END_IF
						ELSE
							arrListOfDevices[byCounterForArray].bNotAllDataIncluded := TRUE;
						END_IF
					//Find the Member Counter Reading
					jsonPropID := fbJsonRead.FindMember(jsonDoc, 'CounterReading');
						IF jsonPropID <> 0 THEN
							IF fbJsonRead.IsNumber(jsonPropID) THEN
								arrListOfDevices[byCounterForArray].lrCounterReading := fbJsonRead.GetDouble(jsonPropID);
									//Limit for 2 commas
									IF arrListOfDevices[byCounterForArray].lrCounterReading >= - 999999999999999 AND arrListOfDevices[byCounterForArray].lrCounterReading <= 999999999999999 THEN
										arrListOfDevices[byCounterForArray].lrCounterReading := LINT_TO_LREAL(LREAL_TO_LINT((arrListOfDevices[byCounterForArray].lrCounterReading) * 100)) / 100;	
									END_IF	
							END_IF
						ELSE
							arrListOfDevices[byCounterForArray].bNotAllDataIncluded := TRUE;
						END_IF
					//Find the Member Counter Reading T1
					jsonPropID := fbJsonRead.FindMember(jsonDoc, 'CounterReadingT1');
						IF jsonPropID <> 0 THEN
							IF fbJsonRead.IsNumber(jsonPropID) THEN
								arrListOfDevices[byCounterForArray].lrCounterReadingT1 := fbJsonRead.GetDouble(jsonPropID);
									//Limit for 2 commas
									IF arrListOfDevices[byCounterForArray].lrCounterReadingT1 >= - 999999999999999 AND arrListOfDevices[byCounterForArray].lrCounterReadingT1 <= 999999999999999 THEN
										arrListOfDevices[byCounterForArray].lrCounterReadingT1 := LINT_TO_LREAL(LREAL_TO_LINT((arrListOfDevices[byCounterForArray].lrCounterReadingT1) * 100)) / 100;	
									END_IF	
							END_IF
						ELSE
							arrListOfDevices[byCounterForArray].bNotAllDataIncluded := TRUE;
						END_IF
					//Find the Member Counter Reading T2
					jsonPropID := fbJsonRead.FindMember(jsonDoc, 'CounterReadingT2');
						IF jsonPropID <> 0 THEN
							IF fbJsonRead.IsNumber(jsonPropID) THEN
								arrListOfDevices[byCounterForArray].lrCounterReadingT2 := fbJsonRead.GetDouble(jsonPropID);
									//Limit for 2 commas
									IF arrListOfDevices[byCounterForArray].lrCounterReadingT2 >= - 999999999999999 AND arrListOfDevices[byCounterForArray].lrCounterReadingT2 <= 999999999999999 THEN
										arrListOfDevices[byCounterForArray].lrCounterReadingT2 := LINT_TO_LREAL(LREAL_TO_LINT((arrListOfDevices[byCounterForArray].lrCounterReadingT2) * 100)) / 100;	
									END_IF	
							END_IF
						ELSE
							arrListOfDevices[byCounterForArray].bNotAllDataIncluded := TRUE;
						END_IF
					//Find the Member Counter Reading T3
					jsonPropID := fbJsonRead.FindMember(jsonDoc, 'CounterReadingT3');
						IF jsonPropID <> 0 THEN
							IF fbJsonRead.IsNumber(jsonPropID) THEN
								arrListOfDevices[byCounterForArray].lrCounterReadingT3 := fbJsonRead.GetDouble(jsonPropID);
									//Limit for 2 commas
									IF arrListOfDevices[byCounterForArray].lrCounterReadingT3 >= - 999999999999999 AND arrListOfDevices[byCounterForArray].lrCounterReadingT3 <= 999999999999999 THEN
										arrListOfDevices[byCounterForArray].lrCounterReadingT3 := LINT_TO_LREAL(LREAL_TO_LINT((arrListOfDevices[byCounterForArray].lrCounterReadingT3) * 100)) / 100;	
									END_IF	
							END_IF
						ELSE
							arrListOfDevices[byCounterForArray].bNotAllDataIncluded := TRUE;
						END_IF
					//Find the Member Counter Reading T4
					jsonPropID := fbJsonRead.FindMember(jsonDoc, 'CounterReadingT4');
						IF jsonPropID <> 0 THEN
							IF fbJsonRead.IsNumber(jsonPropID) THEN
								arrListOfDevices[byCounterForArray].lrCounterReadingT4 := fbJsonRead.GetDouble(jsonPropID);
									//Limit for 2 commas
									IF arrListOfDevices[byCounterForArray].lrCounterReadingT4 >= - 999999999999999 AND arrListOfDevices[byCounterForArray].lrCounterReadingT4 <= 999999999999999 THEN
										arrListOfDevices[byCounterForArray].lrCounterReadingT4 := LINT_TO_LREAL(LREAL_TO_LINT((arrListOfDevices[byCounterForArray].lrCounterReadingT4) * 100)) / 100;	
									END_IF	
							END_IF
						ELSE
							arrListOfDevices[byCounterForArray].bNotAllDataIncluded := TRUE;
						END_IF
					//Find the Member Counter Reading Import
					jsonPropID := fbJsonRead.FindMember(jsonDoc, 'CounterReadingImport');
						IF jsonPropID <> 0 THEN
							IF fbJsonRead.IsNumber(jsonPropID) THEN
								arrListOfDevices[byCounterForArray].lrCounterReadingImp := fbJsonRead.GetDouble(jsonPropID);
									//Limit for 2 commas
									IF arrListOfDevices[byCounterForArray].lrCounterReadingImp >= - 999999999999999 AND arrListOfDevices[byCounterForArray].lrCounterReadingImp <= 999999999999999 THEN
										arrListOfDevices[byCounterForArray].lrCounterReadingImp := LINT_TO_LREAL(LREAL_TO_LINT((arrListOfDevices[byCounterForArray].lrCounterReadingImp) * 100)) / 100;	
									END_IF	
							END_IF
						ELSE
							arrListOfDevices[byCounterForArray].bNotAllDataIncluded := TRUE;
						END_IF
					//Find the Member Counter Reading Export
					jsonPropID := fbJsonRead.FindMember(jsonDoc, 'CounterReadingExport');
						IF jsonPropID <> 0 THEN
							IF fbJsonRead.IsNumber(jsonPropID) THEN
								arrListOfDevices[byCounterForArray].lrCounterReadingExp := fbJsonRead.GetDouble(jsonPropID);
									//Limit for 2 commas
									IF arrListOfDevices[byCounterForArray].lrCounterReadingExp >= - 999999999999999 AND arrListOfDevices[byCounterForArray].lrCounterReadingExp <= 999999999999999 THEN
										arrListOfDevices[byCounterForArray].lrCounterReadingExp := LINT_TO_LREAL(LREAL_TO_LINT((arrListOfDevices[byCounterForArray].lrCounterReadingExp) * 100)) / 100;	
									END_IF	
							END_IF
						ELSE
							arrListOfDevices[byCounterForArray].bNotAllDataIncluded := TRUE;
						END_IF
					//Start with the next Value from the Array
					jsonIteratorArrayStart := fbJsonRead.NextArray(jsonIteratorArrayStart);
			END_WHILE
				bDone := TRUE;
		END_IF
END_IF

END_FUNCTION_BLOCK

// ---- FBs/Suurstoffi Zug/Energy Part/Client FBs/FB_Get_Data_Energy_Surstoffi.TcPOU
{attribute 'hide_all_locals'}
FUNCTION_BLOCK FB_Get_Data_Energy_Surstoffi
VAR_INPUT
	bStart						: BOOL;															//Start the connection to the Service
	sHostname					: STRING(255);													//Hostname or IP Adress from the Energy Service			
END_VAR
VAR_OUTPUT
	bValidResult				: BOOL;															//Valid Result received from Server
    bBusy						: BOOL;															//Function is Busy
    bError						: BOOL;															//Error sucess
	hrErrorCode       			: HRESULT;														//Error Result from Http Client
	arrValuesEnergy				: ARRAY[0..9] OF ST_Values_Energy_Surstoffi;					//Datapoints with Value in a array
END_VAR
VAR
	fbHttpClientEnergyHttp		: FB_IotHttpClient :=(tConnectionTimeout:=T#15S);				//Http Client Function
	fbHttpGet					: FB_HTTP_Get_Energy_Surstoffi;									//Http Get Request to the Energy Service
	fbJson						: FB_Decode_Json_Energy;										//Deconde received Json
	timStartRequest				: TON;															//Timer to Start the Request
	timDissableFunctions		: TON;															//Timer to dissable the Function after Lynus_Standards.Constants_General.tTimeDissableLynusFunctions Days without connection to the Lynus Cloud
	timResetConnectionOnGVL		: TON;															//Timer to try reset the connection Flag on the GVL. (When somebody delete the Connection Function and make only a onlinechange)
	FPStartRequest				: R_TRIG;														//Internal positive Edge
	FNStart						: F_TRIG;														//Internal negative Edge
END_VAR

//Creator : Kai Ebensperger
//Company : Lynus AG
//Date : 18.02.2021
//Version : 1.0.0.0

//With this Function is possible to send a HTTP Get Request to the System in the Surstoffi Area how save the Modbus Energy Data and the Solar Log Energy Data

(*-------------------------------------------------------------Service from Backend is ready and check the connection to backen for dissabel/enable Function---------------------------------------------------------------*)

//Try to reset the variable for connection on the GVL. When all is normal then the Lynus Mqtt connection function set this variable to true in the next cycle
//When we have no connection to the backend then after Lynus_Standards.Constants_General.tTimeDissableLynusFunctions days the Function is dissabled with all of his functionalities
timResetConnectionOnGVL(IN:= NOT timResetConnectionOnGVL.Q, PT:= T#1H, Q=> , ET=> );
	IF timResetConnectionOnGVL.Q THEN Lynus_Standards.GVL_Communicator.bStateConnectionToEnableFunctions := FALSE; END_IF
		IF NOT Lynus_Standards.GVL_Communicator.bStateConnectionToEnableFunctions THEN timDissableFunctions.IN := TRUE; ELSE timDissableFunctions.IN := FALSE; END_IF  
			timDissableFunctions(IN:= , PT:= Lynus_Standards.Constants_General.tTimeDissableLynusFunctions, Q=> , ET=> );

(*------------------------------------------------------------------------------------Configure HTTP Client------------------------------------------------------------------------------------------------------*)

IF NOT fbHttpClientEnergyHttp.bConfigured THEN 
	fbHttpClientEnergyHttp.sHostName := sHostname;
    fbHttpClientEnergyHttp.nHostPort:= 8086;
	fbHttpClientEnergyHttp.stTLS.bNoServerCertCheck:= FALSE;
END_IF

//Timer to start the Request
FPStartRequest(CLK:= bStart, Q=> );
	timStartRequest(IN:= bStart AND NOT timStartRequest.Q AND NOT timDissableFunctions.Q, PT:= T#30S, Q=> , ET=> );
		IF (timStartRequest.Q AND NOT bBusy) OR (FPStartRequest.Q AND NOT bBusy) THEN fbHttpGet.bSend := TRUE; END_IF

//Http Get Function
fbHttpGet(
	bSend:= , 
	tTimeOut:= T#20S,
	fbClient:= fbHttpClientEnergyHttp, 
	bValidResult=> bValidResult, 
	bBusy=> bBusy, 
	bError=> , 
	sContent=> );

fbHttpGet.bSend := FALSE;
	
//Decode Json
fbJson(
	bStart:= bStart AND NOT timDissableFunctions.Q,
	bExecute:= bValidResult, 
	sContent:= fbHttpGet.sContent, 
	bDone=> , 
	bError=> , 
	arrValuesEnergy=> arrValuesEnergy);

//Http Client
FNStart(CLK:= bStart, Q=> );
	IF FNStart.Q THEN fbHttpClientEnergyHttp.Disconnect(); END_IF

fbHttpClientEnergyHttp.Execute();

//Error
IF fbHttpGet.bError OR fbJson.bError OR fbHttpClientEnergyHttp.bError THEN bError := TRUE; ELSE bError := FALSE; END_IF	
	hrErrorCode := fbHttpClientEnergyHttp.hrErrorCode;

END_FUNCTION_BLOCK

// ---- FBs/Suurstoffi Zug/Energy Part/Helper FBs/FB_HTTP_Get_Energy_Surstoffi.TcPOU
{attribute 'hide_all_locals'}
{attribute 'conditionalshow'}
FUNCTION_BLOCK FB_HTTP_Get_Energy_Surstoffi
VAR_INPUT
	{attribute 'hide'}
    bSend           	: BOOL;													//Send the Request
	{attribute 'hide'}
	tTimeOut			: TIME := T#10S;										//Timer for Timeout
END_VAR
VAR_IN_OUT
	{attribute 'hide'}
    fbClient          	: FB_IotHttpClient;										//HTTP Client Data
END_VAR
VAR_OUTPUT
	{attribute 'hide'}
	bValidResult		: BOOL;													//Valid Result received from Server
	{attribute 'hide'}
    bBusy             	: BOOL;													//Function is Busy
	{attribute 'hide'}
    bError           	: BOOL;													//Error sucess
	{attribute 'hide'}
	sContent         	: STRING(7500);											//Received Content
END_VAR
VAR
    fbRequest         	: FB_IotHttpRequest;									//Http Function
	timTimeout			: TON;													//Timer for Timeout
	RisingEdge        	: R_TRIG;												//Internal positive edge
   	bGetContentResult 	: BOOL;													//Get Content Result
	nState				: UDINT;												//Statemaschine
  	nReqCount			: UDINT;												//Counter requests
    nResCount			: UDINT;												//Counter results
    nValidResCount		: UDINT;												//Counter valid results
    nErrCount			: UDINT;												//Error Counter
END_VAR

//Creator : Kai Ebensperger
//Company : Lynus AG
//Date : 18.02.2021
//Version : 1.0.0.0

//With this Function is possible to send a HTTP Get Request to the System in the Surstoffi Area how save the Modbus Energy Data and the Solar Log Energy Data

//Timer for Timeout
timTimeout(IN:= nState = 1 AND bBusy, PT:= tTimeOut, Q=> , ET=> );
	IF timTimeout.Q THEN nState := 0; bBusy := FALSE; END_IF

RisingEdge(CLK:= bSend);

CASE nState OF
0:
    IF RisingEdge.Q THEN
		bValidResult := FALSE;
			IF fbRequest.SendRequest(sUri:= '/query?pretty=true&db=suZEV01&q=SELECT%20%22last%22%28%22Leistung%22%29%20FROM%20%22ZevModbus%22%20WHERE%20%22DPkey%22%3D~%2FSU_18bx_U01_TE01_C001_B890%7CSU_18ax_U01_TE01_C001_B890%7CSU_16xx_U01_TE01_C001_B890%7CSU_20xx_U01_TE01_C001_B890%7CSU_22xx_U01_TE01_C001_B890%7CSU_16xx_U01_TE02_PV00_B890%7CSU_18ax_U01_TE01_PV00_B890%7CSU_18bx_U01_TE01_PV00_B890%7CSU_20xx_U01_TE01_PV00_B890%7CSU_22xx_U01_TE01_PV00_B890%2F%20GROUP%20by%20%22DPkey%22',
									 fbClient:= fbClient, 
									 eRequestType:= ETcIotHttpRequestType.HTTP_Get, 0, 0, 0) THEN
				nState:= 1;
				nReqCount:= nReqCount+1;
				bBusy:= TRUE;
				bError:= FALSE;
			END_IF
    END_IF
1:
    IF NOT fbRequest.bBusy THEN
        bError:= TRUE;
        IF NOT fbRequest.bError THEN
            bGetContentResult:= fbRequest.GetContent(pContent:= ADR(sContent), 
                                                     nContentSize:= SIZEOF(sContent), 
                                                     bSetNullTermination:= TRUE);
            IF fbRequest.nStatusCode >= 200 AND fbRequest.nStatusCode < 300 THEN
                	bValidResult := TRUE;
                    nValidResCount:= nValidResCount+1;
                    bError:= FALSE;
               		nResCount:= nResCount+1;
           END_IF
        END_IF
        nState:= 0;
        bBusy:= FALSE;
        IF bError THEN
            nErrCount:= nErrCount+1;
        END_IF
    END_IF
END_CASE

END_FUNCTION_BLOCK

// ---- FBs/Suurstoffi Zug/Energy Part/Helper FBs/FB_Decode_Json_Energy.TcPOU
{attribute 'hide_all_locals'}
{attribute 'conditionalshow'}
FUNCTION_BLOCK FB_Decode_Json_Energy
VAR_INPUT
	{attribute 'hide'}
	bStart							: BOOL;													//Function is running
	{attribute 'hide'}
	bExecute						: BOOL;													//Start the decoding
	{attribute 'hide'}
	sContent						: STRING(7500);											//Received Content
END_VAR
VAR_OUTPUT
	{attribute 'hide'}
	bDone							: BOOL;													//Function Done
	{attribute 'hide'}
	bError							: BOOL;													//Error Flag
	{attribute 'hide'}
	arrValuesEnergy					: ARRAY[0..9] OF ST_Values_Energy_Surstoffi;			//Datapoints with Value in a array
END_VAR
VAR
	fbJson            				: FB_JsonDomParser;										//Function Json Parser
	FPExecute						: R_TRIG;												//Internal positive edge
	jsonDoc           				: SJsonValue;											//Initila Json Value
	//First Member
	jsonIteratorStartMember1		: SJsonIterator;										//Json Start with 1 Member
	jsonValMember1					: SJsonValue;											//Json Vale from 1 Member
	//First Array
	jsonIteratorStartArray1			: SJsonIterator;										//Json Start with 1 Array
	jsonIteratorEndArray1			: SJsonIterator;										//Json Start with 1 Array	
	jsonValueArray1					: SJsonValue;											//Json Value 1 Array
	jsonValMemberArray1				: SJsonValue;											//Json Value from the last member in 1 Array	
	//Second Array
	jsonIteratorStartArray2			: SJsonIterator;										//Json Start with 2 Array
	jsonIteratorEndArray2			: SJsonIterator;										//Json Start with 2 Array	
	jsonValueArray2					: SJsonValue;											//Json Value 2 Array
	//Member "tags"
	jsonContMemberTags				: SJsonValue;											//Json Value Tags
	jsonValMemberTags				: SJsonValue;											//Json Value Tags
	//Member "columns"
	jsonIteratorStartArrayColumns	: SJsonIterator;										//Json Start with Array columns
	jsonIteratorEndArrayColumns		: SJsonIterator;										//Json Start with Array columns
	jsonContMemberColumns			: SJsonValue;											//Json Value Columns
	jsonValArrayColumns				: SJsonValue;											//Json Value for Array
	//Member "values"
	jsonIteratorStartArrayValues1	: SJsonIterator;										//Json Start with Array 1 Values
	jsonIteratorEndArrayValues1		: SJsonIterator;										//Json Start with Array 1 Values
	jsonIteratorStartArrayValues2	: SJsonIterator;										//Json Start with Array 2 Values
	jsonIteratorEndArrayValues2		: SJsonIterator;										//Json Start with Array 2 Values
	jsonContMemberValues			: SJsonValue;											//Json Value Columns
	jsonValArray1					: SJsonValue;											//Json Value Array 1
	jsonValArray2					: SJsonValue;											//Json Value Array 2
	//Other Variables
	byLoop							: BYTE;													//Loop to clear the Output Array befor insert the new Data
	byCounterColumns1				: BYTE;													//Counter to check on what possiton is the value last or time in the member colums
	byCounterColumns2				: BYTE;													//Counter to fill the Position Values Array that we know on what position we found the time in the next member values
	byCounterColumns3				: BYTE;													//Counter to fill the Position Values Array that we know on what position we found the value in the next member values
	arrCounter						: ARRAY[1..3] OF BYTE;									//Array with counter status to fill the content in the Output array	
	arrPositionTime					: ARRAY[0..9] OF BYTE;									//Save the Position who the Time is saved in the values member array	
	arrPositionValue				: ARRAY[0..9] OF BYTE;									//Save the Position who the value is saved in the values member array									
END_VAR

//Creator : Kai Ebensperger
//Company : Lynus AG
//Date : 18.02.2021
//Version : 1.0.0.0

//With this Fuction is possible to decode the Json String that we received from the Interface from PV soll and the Modbus Counters in the area Surstoffi
//The Message has more Arrays and members included

FPExecute(CLK:= bExecute, Q=> );
	jsonDoc:= fbJson.ParseDocument(sContent);

bDone := FALSE;

IF NOT bStart THEN 
	FOR byLoop := 0 TO 9 BY 1 DO
		arrValuesEnergy[byLoop].sId := '';
			arrValuesEnergy[byLoop].sTimestamp := '';
				arrValuesEnergy[byLoop].lrValue := 0;
	END_FOR
END_IF
	
IF jsonDoc <> 0 AND FPExecute.Q AND bStart THEN

	//Clear Counter
	arrCounter[1] := 0; arrCounter[2] := 0; arrCounter[3] := 0; byCounterColumns1 := 0; byCounterColumns2 := 0; byCounterColumns3 := 0; bError := FALSE;
		//Clear Internal array
		FOR byLoop := 0 TO 9 BY 1 DO
			arrPositionTime[byLoop] := 0;
				arrPositionValue[byLoop] := 0;	
		END_FOR
			//Clear Output Array
			FOR byLoop := 0 TO 9 BY 1 DO
				arrValuesEnergy[byLoop].sId := '';
					arrValuesEnergy[byLoop].sTimestamp := '';
						arrValuesEnergy[byLoop].lrValue := 0;
			END_FOR
	
//Start with the first Member and get this value
jsonIteratorStartMember1 := fbJson.MemberBegin(jsonDoc);
	jsonValMember1 := fbJson.GetMemberValue(jsonIteratorStartMember1);	

	
//Start to decode 1 Array content with the member "series"	
jsonIteratorStartArray1 := fbJson.ArrayBegin(jsonValMember1);
jsonIteratorEndArray1 := fbJson.ArrayEnd(jsonValMember1);
	WHILE jsonIteratorStartArray1 <> jsonIteratorEndArray1 DO
		jsonValueArray1 := fbJson.GetArrayValue(jsonIteratorStartArray1);
			jsonValMemberArray1 := fbJson.FindMember(jsonValueArray1,'series');	
				jsonIteratorStartArray1 := fbJson.NextArray(jsonIteratorStartArray1);
	END_WHILE

	//Start to decode 2 Array content
	IF jsonValMemberArray1 <> 0 THEN
		jsonIteratorStartArray2 := fbJson.ArrayBegin(jsonValMemberArray1);
		jsonIteratorEndArray2 := fbJson.ArrayEnd(jsonValMemberArray1);
			WHILE jsonIteratorStartArray2 <> jsonIteratorEndArray2 DO
				jsonValueArray2 := fbJson.GetArrayValue(jsonIteratorStartArray2);
					//Member "Tags"
					jsonContMemberTags := fbJson.FindMember(jsonValueArray2,'tags');
						IF jsonContMemberTags <> 0 THEN
							//Find the member "DPkey"
							jsonValMemberTags := fbJson.FindMember(jsonContMemberTags,'DPkey');
								IF jsonValMemberTags <> 0 AND fbJson.IsString(jsonValMemberTags) THEN
									IF arrCounter[1] > 9 THEN bError := TRUE; END_IF
										arrCounter[1] := LIMIT(0,arrCounter[1],9);
											arrValuesEnergy[arrCounter[1]].sID := fbJson.GetString(jsonValMemberTags);
												arrCounter[1] := arrCounter[1] + 1;	
								END_IF 
						END_IF 
					//Member "columns"
					jsonContMemberColumns := fbJson.FindMember(jsonValueArray2,'columns');
						IF jsonContMemberColumns <> 0 THEN
							jsonIteratorStartArrayColumns := fbJson.ArrayBegin(jsonContMemberColumns);
							jsonIteratorEndArrayColumns := fbJson.ArrayEnd(jsonContMemberColumns);	
								WHILE jsonIteratorStartArrayColumns <> jsonIteratorEndArrayColumns DO
									jsonValArrayColumns := fbJson.GetArrayValue(jsonIteratorStartArrayColumns);
										IF jsonValArrayColumns <> 0 AND fbJson.IsString(jsonValArrayColumns) THEN  
											//Find the time text in the json string
											IF fbJson.GetString(jsonValArrayColumns) = 'time' THEN
												IF byCounterColumns2 > 9 THEN bError := TRUE; EXIT; END_IF
													byCounterColumns2 := LIMIT(0,byCounterColumns2,9);	
														arrPositionTime[byCounterColumns2] := byCounterColumns1;
															byCounterColumns2 := byCounterColumns2 + 1;
											END_IF 
												//Find the last text in the json string
												IF fbJson.GetString(jsonValArrayColumns) = 'last' THEN
													IF byCounterColumns3 > 9 THEN bError := TRUE; EXIT; END_IF
														byCounterColumns3 := LIMIT(0,byCounterColumns3,9);
															arrPositionValue[byCounterColumns3] := byCounterColumns1;
																byCounterColumns3 := byCounterColumns3 + 1;
													END_IF
										END_IF
											byCounterColumns1 := byCounterColumns1 + 1;
												IF byCounterColumns1 > 250 THEN bError := TRUE; EXIT; END_IF
													jsonIteratorStartArrayColumns := fbJson.NextArray(jsonIteratorStartArrayColumns);
								END_WHILE   
									byCounterColumns1 := 0;
						END_IF 
					//Member "values"
					jsonContMemberValues := fbJson.FindMember(jsonValueArray2,'values');
						IF jsonContMemberValues <> 0 THEN
							//Decode first Array
						 	jsonIteratorStartArrayValues1 := fbJson.ArrayBegin(jsonContMemberValues);
							jsonIteratorEndArrayValues1 := fbJson.ArrayEnd(jsonContMemberValues);
								WHILE jsonIteratorStartArrayValues1 <> jsonIteratorEndArrayValues1 DO
									jsonValArray1 :=  fbJson.GetArrayValue(jsonIteratorStartArrayValues1);
										//Decode second Array
										IF jsonValArray1 <> 0 THEN 
											jsonIteratorStartArrayValues2 := fbJson.ArrayBegin(jsonValArray1);
											jsonIteratorEndArrayValues2 := fbJson.ArrayEnd(jsonValArray1);	
												WHILE jsonIteratorStartArrayValues2 <> jsonIteratorEndArrayValues2 DO
													jsonValArray2 := fbJson.GetArrayValue(jsonIteratorStartArrayValues2);
														//Find the Timestamp
														IF jsonValArray2 <> 0 AND fbJson.IsString(jsonValArray2) THEN
															IF arrCounter[2] > 9 THEN bError := TRUE; END_IF
																arrCounter[2] := LIMIT(0,arrCounter[2],9);
																	arrValuesEnergy[arrCounter[2]].sTimestamp := fbJson.GetString(jsonValArray2);
																		arrCounter[2] := arrCounter[2] + 1;	
														END_IF  
														//Find the Value
														IF jsonValArray2 <> 0 AND fbJson.IsNumber(jsonValArray2) THEN
															IF arrCounter[3] > 9 THEN bError := TRUE; END_IF
																arrCounter[3] := LIMIT(0,arrCounter[3],9);
																	IF fbJson.IsDouble(jsonValArray2) THEN arrValuesEnergy[arrCounter[3]].lrValue := fbJson.GetDouble(jsonValArray2); END_IF
																	IF fbJson.IsInt64(jsonValArray2) THEN arrValuesEnergy[arrCounter[3]].lrValue := LINT_TO_LREAL(fbJson.GetInt64(jsonValArray2)); END_IF
																	IF fbJson.IsUint64(jsonValArray2) THEN arrValuesEnergy[arrCounter[3]].lrValue := ULINT_TO_LREAL(fbJson.GetUint64(jsonValArray2)); END_IF 	
																		arrCounter[3] := arrCounter[3] + 1;
														END_IF 
													jsonIteratorStartArrayValues2 := fbJson.NextArray(jsonIteratorStartArrayValues2);	
												END_WHILE
										END_IF
									jsonIteratorStartArrayValues1 := fbJson.NextArray(jsonIteratorStartArrayValues1);
								END_WHILE	
						END_IF		
				jsonIteratorStartArray2 := fbJson.NextArray(jsonIteratorStartArray2);
			END_WHILE
	END_IF
	
	//Limit for 2 Commas and convert to KW
	FOR byLoop := 0 TO 9 BY 1 DO
		arrValuesEnergy[byLoop].lrValue := arrValuesEnergy[byLoop].lrValue / 1000;
			arrValuesEnergy[byLoop].lrValue := LINT_TO_LREAL(LREAL_TO_LINT(arrValuesEnergy[byLoop].lrValue * 100)) / 100;
	END_FOR
	
	//Done
	IF NOT bError THEN bDone := TRUE; END_IF
	
END_IF

END_FUNCTION_BLOCK

// ---- FBs/Suurstoffi Zug/Iosys Part/Client FBs/FB_Get_Data_Iosys.TcPOU
{attribute 'hide_all_locals'}
FUNCTION_BLOCK FB_Get_Data_Iosys
VAR_INPUT
	bStart						: BOOL;															//Start the connection to the Aprol Server
	byQuantity					: BYTE;															//Quantity of Datapoints
	sHostname					: STRING(255);													//Hostname or IP Adress from the Aprol Server
	sProjectname				: STRING(30);													//Projectname
	sRuntimeSystem				: STRING(30);													//Name from the Runtime System
	tWaitTimeTokenMode			: TIME := T#5S;													//Time to wait after new request if Token mode is active
	arrListDatapoints			: ARRAY[0..249] OF STRING(38);									//List with all the Datapoints
END_VAR
VAR_OUTPUT
	bValidResult				: BOOL;															//Valid Result received from Server
    bBusy						: BOOL;															//Function is Busy
    bError						: BOOL;															//Error sucess
	hrErrorCode       			: HRESULT;														//Error Result from Http Client
	sToken		      			: STRING(255);													//Last Token from the content
	arrValuesIosys				: ARRAY[0..249] OF ST_Values_Checked_Iosys;						//Datapoints with Value in a array
END_VAR
VAR
	fbHttpClientIosysHttp		: FB_IotHttpClient :=(tConnectionTimeout:=T#15S);				//Http Client Function
	fbHttpGet					: FB_HTTP_Get_Iosys;											//Http Get Request to the Aprol Server
	fbJson						: FB_Decode_Json_Iosys;											//Deconde received Json
	fbCheckList					: FB_Check_List_Iosys;											//Function to Update the Values
	FPStart						: R_TRIG;														//Intern positive edge
	FPError						: R_TRIG;														//Intern positive edge
	FPResult					: R_TRIG;														//Intern positive edge
	FNStart						: F_TRIG;														//Internal negative Edge
	timValidResult				: TON;															//Timer to wait for valid result
	timRestart					: TON;															//Timer to restart the function after error
	timWaitStep3				: TON;															//Timer to wait in Step 3 before make new Request
	timDissableFunctions		: TON;															//Timer to dissable the Function after Lynus_Standards.Constants_General.tTimeDissableLynusFunctions Days without connection to the Lynus Cloud
	timResetConnectionOnGVL		: TON;															//Timer to try reset the connection Flag on the GVL. (When somebody delete the Connection Function and make only a onlinechange)
	bErrorValidResult			: BOOL;															//No valid Data received
	byWaitInStep				: BYTE;															//Cycles to wait in Step
	uiState						: UINT;															//Statemaschine
END_VAR

//Creator : Kai Ebensperger
//Company : Lynus AG
//Date : 02.02.2021
//Version : 1.0.0.0

//With this Function Block its possible to read out Data from a Aprol Server over the Iosys Interface
//The first Request is a Request with all Datapoints from the Input Array. 
//After sucess, we receive a Token from the Server. After that, the PLC Function switch in the Token Mode.
//The request to the Server work then with the reveiced Token and not wiht the list of eacht Datapoint. 
//If we stop the Communication or a Error Sucess, the Function start with first Request with all datapoints and switch then again in the Token mode. 
//The Token has a validity from 10 seconds.

//Examples for the 2 Modes for Request
//REQUEST 1
//10.1.31.8/iosys/Suurstoffi/ASRO02/json/get?id=SU_16xx_U01_TC02_L002_B800_M01.ha; OR =>
//For more Variablen use id=SU_16xx_U01_TC02_L002_B800_M01.ha,SU_16xx_U01_TC02_L002_B850_M01.ha;
//REQUEST 2
//Token
//10.1.31.8/iosys/Suurstoffi/ASRO02/json/get?token=wlEtAw0fKrK&req=2;

(*-------------------------------------------------------------Service from Backend is ready and check the connection to backen for dissabel/enable Function---------------------------------------------------------------*)

//Try to reset the variable for connection on the GVL. When all is normal then the Lynus Mqtt connection function set this variable to true in the next cycle
//When we have no connection to the backend then after Lynus_Standards.Constants_General.tTimeDissableLynusFunctions days the Function is dissabled with all of his functionalities
timResetConnectionOnGVL(IN:= NOT timResetConnectionOnGVL.Q, PT:= T#1H, Q=> , ET=> );
	IF timResetConnectionOnGVL.Q THEN Lynus_Standards.GVL_Communicator.bStateConnectionToEnableFunctions := FALSE; END_IF
		IF NOT Lynus_Standards.GVL_Communicator.bStateConnectionToEnableFunctions THEN timDissableFunctions.IN := TRUE; ELSE timDissableFunctions.IN := FALSE; END_IF  
			timDissableFunctions(IN:= , PT:= Lynus_Standards.Constants_General.tTimeDissableLynusFunctions, Q=> , ET=> );

(*------------------------------------------------------------------------------------Configure HTTP Client------------------------------------------------------------------------------------------------------*)

IF NOT fbHttpClientIosysHttp.bConfigured THEN 
	fbHttpClientIosysHttp.sHostName := sHostname;
    fbHttpClientIosysHttp.nHostPort:= 80;
	fbHttpClientIosysHttp.stTLS.bNoServerCertCheck:= FALSE;
END_IF

//Min and Max Value
tWaitTimeTokenMode := LIMIT(T#0S,tWaitTimeTokenMode,T#10S);

//Start
FPStart(CLK:= bStart, Q=> );
	IF FPStart.Q AND fbHttpClientIosysHttp.bConfigured AND NOT bBusy THEN uiState := 1; END_IF
		
//Stop	
IF NOT bStart OR timDissableFunctions.Q THEN uiState := 0; END_IF	

CASE uiState OF
	
	0://Init
		fbHttpGet.bSend := FALSE;
			fbHttpGet.bTokenMode := FALSE;
				fbHttpGet.sToken := '';
					fbJson.bExecute := FALSE;
						timValidResult.IN := FALSE;
							timRestart.IN := FALSE;
								byWaitInStep := 0;
									timWaitStep3.IN := FALSE;
					
	1://Start
		fbHttpGet.bSend := TRUE;
			timValidResult.IN := TRUE;
			
		//Next Step	
		IF FPResult.Q AND NOT FPError.Q THEN uiState := 2; timValidResult.IN := FALSE; fbHttpGet.bSend := FALSE; END_IF 
		
		//Error
		IF FPError.Q OR timValidResult.Q THEN uiState := 300; END_IF

	2://Check Json and the Content
		fbJson.bExecute := TRUE;
		
		byWaitInStep := byWaitInStep + 1;
		
		//Next Step
		IF fbJson.bDone THEN fbJson.bExecute := FALSE; uiState := 3; byWaitInStep := 0; END_IF
		
		//No Data encodet
		IF NOT fbJson.bDone AND byWaitInStep >= 2 THEN uiState := 300; END_IF
		
	3://Switch to Token Mode and make Request
		timWaitStep3.IN := TRUE;
	
		IF timWaitStep3.Q THEN
			fbHttpGet.bTokenMode := TRUE;
				fbHttpGet.sToken := sToken;
					fbHttpGet.bSend := TRUE;
						timValidResult.IN := TRUE;
		END_IF
					
		//Next Step	
		IF FPResult.Q AND NOT FPError.Q THEN uiState := 2; timValidResult.IN := FALSE; fbHttpGet.bSend := FALSE; bErrorValidResult := FALSE; timWaitStep3.IN := FALSE; END_IF 
		
		//Error
		IF FPError.Q OR timValidResult.Q THEN uiState := 300; END_IF			
		
	300://Error
	 	bErrorValidResult := TRUE;
			timRestart.IN := TRUE;
				fbHttpGet.bSend := FALSE;
					fbHttpGet.bTokenMode := FALSE;
						fbHttpGet.sToken := '';
							fbJson.bExecute := FALSE;
								timValidResult.IN := FALSE;
									byWaitInStep := 0;
										timWaitStep3.IN := FALSE;
							
		//After Error Wait for new Request
		IF timRestart.Q THEN uiState := 1; timRestart.IN := FALSE; END_IF

END_CASE

//Http Get Request
fbHttpGet(
	bSend:= , 
	bTokenMode:= , 
	byQuantity:= byQuantity, 
	sToken:= , 
	sProjectname:= sProjectname, 
	sRuntimeSystem:= sRuntimeSystem, 
	tTimeOut:= T#20S,
	arrListDatapoints:= arrListDatapoints, 
	fbClient:= fbHttpClientIosysHttp, 
	bValidResult=> bValidResult, 
	bBusy=> bBusy, 
	bError=> , 
	sContent=> );

FPResult(CLK:= bValidResult, Q=> );	
	
FPError(CLK:= fbHttpGet.bError, Q=> );	

//Json Decode Function
fbJson(bExecute:= , sContent:= fbHttpGet.sContent, sToken=> sToken, arrValuesIosys=> , bDone=> );	

//Check the Datapoints
fbCheckList(
	bStart:= bStart AND NOT timDissableFunctions.Q, 
	bValidResult:= bValidResult, 
	bDone:= fbJson.bDone, 
	arrValuesIosys:= fbJson.arrValuesIosys, 
	arrCheckedValues=> arrValuesIosys);

//Http Client
FNStart(CLK:= bStart, Q=> );
	IF FNStart.Q THEN fbHttpClientIosysHttp.Disconnect(); END_IF

fbHttpClientIosysHttp.Execute();

//Set/reset Error bit
IF fbHttpGet.bError OR bErrorValidResult OR fbHttpClientIosysHttp.bError THEN bError := TRUE; ELSE bError := FALSE; END_IF
	hrErrorCode := fbHttpClientIosysHttp.hrErrorCode;	

//Timer to check valid result
timValidResult(IN:= , PT:= T#11S, Q=> , ET=> );

//Timer to resart the Function after Error
timRestart(IN:= , PT:= T#10S, Q=> , ET=> );

//Timer Step 3
timWaitStep3(IN:= , PT:= tWaitTimeTokenMode, Q=> , ET=> );

END_FUNCTION_BLOCK

// ---- FBs/Suurstoffi Zug/Iosys Part/Helper FBs/FB_HTTP_Get_Iosys.TcPOU
{attribute 'hide_all_locals'}
{attribute 'conditionalshow'}
FUNCTION_BLOCK FB_HTTP_Get_Iosys
VAR_INPUT
	{attribute 'hide'}
    bSend				: BOOL;													//Send the Request
	{attribute 'hide'}
	bTokenMode			: BOOL;													//Make the Request with the Token
	{attribute 'hide'}
	byQuantity			: BYTE;													//Quantity of Datapoints
	{attribute 'hide'}
	sToken		      	: STRING(255);											//Token for the Request
	{attribute 'hide'}
	sProjectname		: STRING(30);											//Projectname
	{attribute 'hide'}
	sRuntimeSystem		: STRING(30);											//Name from the Runtime System
	{attribute 'hide'}
	tTimeOut			: TIME := T#10S;										//Timer for Timeout
	{attribute 'hide'}
	arrListDatapoints	: ARRAY[0..249] OF STRING(38);							//List with all the Datapoints
END_VAR
VAR_IN_OUT
	{attribute 'hide'}
    fbClient			: FB_IotHttpClient;										//HTTP Client Data
END_VAR
VAR_OUTPUT
	{attribute 'hide'}
	bValidResult		: BOOL;													//Valid Result received from Server
	{attribute 'hide'}
    bBusy				: BOOL;													//Function is Busy
	{attribute 'hide'}
    bError				: BOOL;													//Error sucess
	{attribute 'hide'}
	sContent			: STRING(35000);										//Received Content
END_VAR
VAR
    fbRequest			: FB_IotHttpRequest;									//Http Function
	timTimeout			: TON;													//Timer for Timeout
	RisingEdge			: R_TRIG;												//Internal positive edge
	bGetContentResult	: BOOL;													//Get Content Result	
	byLoop				: BYTE;													//Variable foor Loop to prepear the URI
    nState				: UDINT;												//Statemaschine
  	nReqCount			: UDINT;												//Counter requests
    nResCount			: UDINT;												//Counter results
    nValidResCount		: UDINT;												//Counter valid results
    nErrCount			: UDINT;												//Error Counter
	sUriStart			: STRING(81);											//Start URI
	sUriComplete		: STRING(10000);										//Complete URI
END_VAR

//Creator : Kai Ebensperger
//Company : Lynus AG
//Date : 02.02.2021
//Version : 1.0.0.0

//With this Fuction is possible to send a HTTP Get Request to the Iosys Interface from the Aprol Server from the B&R Company.
//To make a  requerst to the right Project, the Projectname and the Ruhntime System is necessary.
//In the Input Array you can insert all Datapoint with rifht Name from the System form what do you want the Values
//The Request can send with each Datapoint. Then The Token Mode is disabled
//Its also possible to use the Token Mode. To use this, make first the Request with all Datapoitns that are needed to the API. With the Response you received a Token.
//With this Token then you can make within 10 seconds a Request and you receive all Datapoint from the first Request.

//Timer for Timeout
timTimeout(IN:= nState = 1 AND bBusy, PT:= tTimeOut, Q=> , ET=> );
	IF timTimeout.Q THEN nState := 0; bBusy := FALSE; END_IF

byQuantity := LIMIT(0,byQuantity,249);

RisingEdge(CLK:= bSend);

CASE nState OF
0:
	IF RisingEdge.Q THEN
		//Prepear URI
		IF NOT bTokenMode THEN
			sUriComplete := '';
				sUriStart := CONCAT(CONCAT('/iosys/',sProjectname),CONCAT(CONCAT('/',sRuntimeSystem),'/json/get?id='));
					sUriComplete := sUriStart;
						FOR byLoop := 0 TO byQuantity BY 1 DO
							CONCAT2(ADR(sUriComplete),ADR(arrListDatapoints[byLoop]),ADR(sUriComplete),SIZEOF(sUriComplete));
								IF byLoop < (byQuantity - 1) THEN CONCAT2(ADR(sUriComplete),ADR(','),ADR(sUriComplete),SIZEOF(sUriComplete)); END_IF	
						END_FOR
							CONCAT2(ADR(sUriComplete),ADR(';'),ADR(sUriComplete),SIZEOF(sUriComplete));		
		ELSE
			sUriComplete := '';
				sUriStart := CONCAT(CONCAT('/iosys/',sProjectname),CONCAT(CONCAT('/',sRuntimeSystem),'/json/get?token='));
					sUriComplete := CONCAT(CONCAT(sUriStart,sToken),';');			
		END_IF

		bValidResult := FALSE;
			
			IF fbRequest.SendRequest(sUri:= sUriComplete,
									 fbClient:= fbClient, 
										eRequestType:= ETcIotHttpRequestType.HTTP_Get, 0, 0, 0) THEN
				nState:= 1;
				nReqCount:= nReqCount+1;
				bBusy:= TRUE;
				bError:= FALSE;
			END_IF
    END_IF
1:
    IF NOT fbRequest.bBusy THEN
        bError:= TRUE;
        IF NOT fbRequest.bError THEN
            bGetContentResult:= fbRequest.GetContent(pContent:= ADR(sContent), 
                                                     nContentSize:= SIZEOF(sContent), 
                                                     bSetNullTermination:= TRUE);
            IF fbRequest.nStatusCode >= 200 AND fbRequest.nStatusCode < 300 THEN
				bValidResult := TRUE;
				bError := FALSE;
				nValidResCount:= nValidResCount+1;
               	nResCount:= nResCount+1;
            END_IF
        END_IF
        nState:= 0;
        bBusy:= FALSE;
        IF bError THEN
            nErrCount:= nErrCount+1;
        END_IF
    END_IF
END_CASE

END_FUNCTION_BLOCK

// ---- FBs/Suurstoffi Zug/Iosys Part/Helper FBs/FB_Decode_Json_Iosys.TcPOU
{attribute 'hide_all_locals'}
{attribute 'conditionalshow'}
FUNCTION_BLOCK FB_Decode_Json_Iosys
VAR_INPUT
	{attribute 'hide'}
	bExecute				: BOOL;										//Start the decoding
	{attribute 'hide'}
	sContent				: STRING(35000);							//Received Content
END_VAR
VAR_OUTPUT
	{attribute 'hide'}
	bDone					: BOOL;										//Function Done
	{attribute 'hide'}
	sToken		      		: STRING(255);								//Last Token from the content
	{attribute 'hide'}
	arrValuesIosys			: ARRAY[0..249] OF ST_Values_Iosys;			//Datapoints with Value in a array
END_VAR
VAR
	fbJson            		: FB_JsonDomParser;							//Function Json Parser
	FPExecute				: R_TRIG;									//Internal positive edge
	jsonDoc           		: SJsonValue;								//Initila Json Value							
	//First Array
	jsonIteratorStartA1		: SJsonIterator;							//Json Start Ilaterator from the 1 Array
	jsonIteratorEndA1		: SJsonIterator;							//Json End Ilaterator from the 1 Array
	jsonValA1_A2         	: SJsonValue;								//Json Value to Get Array Value
	jsonValA1_1         	: SJsonValue;								//Json Value to find Member for the token
	uiCounter				: UINT;										//Counter to find Values in 1 and 2 Array from received Json
	//Second Array 1 Loop to get Array Value
	jsonIteratorStartA2_1	:  SJsonIterator;							//Json Start Ilaterator from the 2 Array to check all Members
	jsonIteratorEndA2_1		:  SJsonIterator;							//Json End Ilaterator from the 2 Array to check all Members
	//Second Array 2 Loop to get Member value
	jsonIteratorStartA2_2	: SJsonIterator;							//Json Start Ilaterator from the 2 Array to check all Values from the necessary Members
	jsonIteratorEndA2_2		: SJsonIterator;							//Json End Ilaterator from the 2 Array to check all Values from the necessary Members
	jsonValA2_1         	: SJsonValue;								//Json Value to Get Array Value
	jsonValA2_2        		: SJsonValue;								//Json Value to Get the Member Value
	byLoop					: BYTE;										//Loop to clear the Output Array befor insert the new Data
	uiCounterArray			: UINT;										//Counter to fill the Values in the Output Array
	sMember					: STRING(255);								//String with the member name
END_VAR

//Creator : Kai Ebensperger
//Company : Lynus AG
//Date : 02.02.2021
//Version : 1.0.0.0

//With this Fuction is possible to decode the Json String that we received from the Iosys Interface from the Aprol Server from the B&R Comapny
//The Message arrives allwas in 2 Arrays. In the 1 Array is the Token from the last request. In the 2 Array all Datapoints with the Values from the Request

FPExecute(CLK:= bExecute, Q=> );
	jsonDoc:= fbJson.ParseDocument(sContent);
		uiCounter := 0;
			uiCounterArray := 0;

bDone := FALSE;
	
IF jsonDoc <> 0 AND FPExecute.Q THEN
	
	//Clear Array
	FOR byLoop := 0 TO 249 BY 1 DO
		arrValuesIosys[byLoop].sId := '';
			arrValuesIosys[byLoop].sTimestamp := '';
				arrValuesIosys[byLoop].sValue := '';
					arrValuesIosys[byLoop].bNoValue := FALSE;	
	END_FOR

jsonIteratorStartA1 := fbJson.ArrayBegin(jsonDoc);
jsonIteratorEndA1 := fbJson.ArrayEnd(jsonDoc);
	//Check the first Array with the token
	WHILE jsonIteratorStartA1 <> jsonIteratorEndA1 DO
		uiCounter := uiCounter + 1;
		jsonValA1_A2 := fbJson.GetArrayValue(jsonIteratorStartA1);
			IF uiCounter = 1 AND fbJson.HasMember(jsonValA1_A2,'token') AND jsonValA1_A2 <> 0 THEN 
				jsonValA1_1 := fbJson.FindMember(jsonValA1_A2,'token'); 
				IF jsonValA1_1 <> 0 AND fbJson.IsString(jsonValA1_1) THEN sToken := fbJson.GetString(jsonValA1_1); END_IF
			END_IF
				IF uiCounter = 2 THEN 
					jsonIteratorStartA2_1 := fbJson.ArrayBegin(jsonValA1_A2);
					jsonIteratorEndA2_1 := fbJson.ArrayEnd(jsonValA1_A2);
						//Check the second Array to parse all menbers 
						WHILE jsonIteratorStartA2_1 <> jsonIteratorEndA2_1 DO
							jsonValA2_1 := fbJson.GetArrayValue(jsonIteratorStartA2_1);	
								IF jsonValA2_1 <> 0 THEN
									jsonIteratorStartA2_2 := fbJson.MemberBegin(jsonValA2_1);
									jsonIteratorEndA2_2 := fbJson.MemberEnd(jsonValA2_1);
										//Check necessary member in Second Array for the values
										WHILE jsonIteratorStartA2_2 <> jsonIteratorEndA2_2 DO
											sMember := fbJson.GetMemberName(jsonIteratorStartA2_2);
												IF sMember = 'ts' THEN 
													jsonValA2_2 := fbJson.GetMemberValue(jsonIteratorStartA2_2); 
														IF fbJson.IsString(jsonValA2_2) AND jsonValA2_2 <> 0 THEN arrValuesIosys[uiCounterArray].sTimestamp := fbJson.GetString(jsonValA2_2); END_IF
												END_IF
												IF sMember = 'id' THEN 
													jsonValA2_2 := fbJson.GetMemberValue(jsonIteratorStartA2_2); 
														IF fbJson.IsString(jsonValA2_2) AND jsonValA2_2 <> 0 THEN arrValuesIosys[uiCounterArray].sId := fbJson.GetString(jsonValA2_2); END_IF
												END_IF
												IF sMember = 'val' THEN 
													jsonValA2_2 := fbJson.GetMemberValue(jsonIteratorStartA2_2); 
														IF fbJson.IsString(jsonValA2_2) AND jsonValA2_2 <> 0 THEN arrValuesIosys[uiCounterArray].sValue := fbJson.GetString(jsonValA2_2); END_IF
												END_IF
													jsonIteratorStartA2_2 := fbJson.NextMember(jsonIteratorStartA2_2);
										END_WHILE
											IF arrValuesIosys[uiCounterArray].sValue = '' THEN arrValuesIosys[uiCounterArray].bNoValue := TRUE; END_IF
											uiCounterArray := uiCounterArray + 1;
												uiCounterArray := LIMIT(0,uiCounterArray,249);
								END_IF
								jsonIteratorStartA2_1 := fbJson.NextArray(jsonIteratorStartA2_1);
						END_WHILE
					END_IF
			jsonIteratorStartA1 := fbJson.NextArray(jsonIteratorStartA1);
	END_WHILE
	//If min the token is received then the function is done
	IF sToken <> '' THEN bDone := TRUE;	END_IF			
END_IF

END_FUNCTION_BLOCK

// ---- FBs/Suurstoffi Zug/Iosys Part/Helper FBs/FB_Check_List_Iosys.TcPOU
{attribute 'hide_all_locals'}
{attribute 'conditionalshow'}
FUNCTION_BLOCK FB_Check_List_Iosys
VAR_INPUT
	{attribute 'hide'}
	bStart						: BOOL;															//Start the Function. False = The Data in the output Array is deleted 
	{attribute 'hide'}
	bValidResult				: BOOL;															//Valid Result received from Server
	{attribute 'hide'}
	bDone						: BOOL;															//Data in Input Array is complete
	{attribute 'hide'}
	arrValuesIosys				: ARRAY[0..249] OF ST_Values_Iosys;								//Datapoints with Value in a array
END_VAR
VAR_OUTPUT
	{attribute 'hide'}
	arrCheckedValues			: ARRAY[0..249] OF ST_Values_Checked_Iosys;						//All Datapoints what are receved from the Server	
END_VAR
VAR
	FPDone						: R_TRIG;														//Internal positive edge
	FNStart						: F_TRIG;														//Internal negative Edge
	bExist						: BOOL;															//Show that the Value just exist in the output Array
	byLPArray					: BYTE;															//Variable for Loop
	byLPArrayIntern				: BYTE;															//Variable for Loop
	byPlaceInArrayInUse			: BYTE;															//Show how much places in the output array are just in use
	byCounterLoop				: BYTE;															//Counter Variable for Loop
	iStateCheckValue			: INT;															//Variable for Statemaschine
	sValue						: STRING(30);													//Value as Strin after preparetion
END_VAR

//Creator : Kai Ebensperger
//Company : Lynus AG
//Date : 17.02.2021
//Version : 1.0.0.0

//Since only the values that have changed are delivered when querying the data points via the token, 
//the values that have not changed but have already occurred must be saved. So that they are not overwritten with 0.

//---------------------------------------------------------------------------Start and Stop the function--------------------------------------------------------------

FNStart(CLK:= bStart, Q=> );
	FPDone(CLK:= bDone, Q=> );

//Start new Session	
IF FPDone.Q AND bValidResult AND bStart AND iStateCheckValue = 0 THEN iStateCheckValue := 1; END_IF
	//Stop
	IF FNStart.Q THEN 
		iStateCheckValue := 0; byPlaceInArrayInUse := 0; sValue := ''; byCounterLoop := 0;	
			//Clear the Output Array
			FOR byLPArray := 0 TO 249 BY 1 DO
				arrCheckedValues[byLPArray].lrValue := 0;
					arrCheckedValues[byLPArray].sId := '';
						arrCheckedValues[byLPArray].sTimestamp := '';	
			END_FOR	
	END_IF
	
//---------------------------------------------------------------------------State Maschine--------------------------------------------------------------

CASE iStateCheckValue OF
	
	1://Write all Variabes to Output
		FOR byLPArray := 0 TO 249 BY 1 DO
			IF arrValuesIosys[byLPArray].sId <> '' AND NOT arrValuesIosys[byLPArray].bNoValue THEN
				arrCheckedValues[byPlaceInArrayInUse].sTimestamp := arrValuesIosys[byLPArray].sTimestamp;
					arrCheckedValues[byPlaceInArrayInUse].sId := arrValuesIosys[byLPArray].sId;
						//Prepear the String Value
						IF FIND(arrValuesIosys[byLPArray].sValue,'.') <> 0 THEN
							sValue := MID(arrValuesIosys[byLPArray].sValue,FIND(arrValuesIosys[byLPArray].sValue,'.') + 2,1);
								arrCheckedValues[byPlaceInArrayInUse].lrValue := STRING_TO_LREAL(sValue);
									//Limit to 2 commas
									arrCheckedValues[byPlaceInArrayInUse].lrValue := LINT_TO_LREAL(LREAL_TO_LINT(arrCheckedValues[byPlaceInArrayInUse].lrValue * 100)) / 100;	
						ELSE
							sValue := MID(arrValuesIosys[byLPArray].sValue,30,1);
								arrCheckedValues[byPlaceInArrayInUse].lrValue := STRING_TO_LREAL(sValue);
						END_IF	
							byPlaceInArrayInUse := byPlaceInArrayInUse + 1;	
								byPlaceInArrayInUse := LIMIT(0,byPlaceInArrayInUse,250);	 
			END_IF
				//All vaiables insert and go to next step
				IF LEN(arrValuesIosys[byLPArray].sId) = 0 OR byPlaceInArrayInUse >= 250 THEN iStateCheckValue := 2; EXIT; END_IF 	
		END_FOR		
 
	2://Wait for new Values
		IF byPlaceInArrayInUse > 249 THEN byPlaceInArrayInUse := 249; END_IF 
			IF FPDone.Q AND bValidResult AND bStart THEN iStateCheckValue := 3; byCounterLoop := 0; END_IF
		
	3://Check the changes
		FOR byLPArray := 0 TO byPlaceInArrayInUse BY 1 DO
			FOR byLPArrayIntern := 0 TO byPlaceInArrayInUse BY 1 DO
				IF arrValuesIosys[byLPArray].sId = arrCheckedValues[byLPArrayIntern].sId THEN
					arrCheckedValues[byLPArrayIntern].sTimestamp := arrValuesIosys[byLPArray].sTimestamp;
						//Prepear the String Value
						IF FIND(arrValuesIosys[byLPArray].sValue,'.') <> 0 THEN
							sValue := MID(arrValuesIosys[byLPArray].sValue,FIND(arrValuesIosys[byLPArray].sValue,'.') + 2,1);
								arrCheckedValues[byLPArrayIntern].lrValue := STRING_TO_LREAL(sValue);
									//Limit to 2 commas
									arrCheckedValues[byLPArrayIntern].lrValue := LINT_TO_LREAL(LREAL_TO_LINT(arrCheckedValues[byLPArrayIntern].lrValue * 100)) / 100;	
						ELSE
							sValue := MID(arrValuesIosys[byLPArray].sValue,30,1);
								arrCheckedValues[byLPArrayIntern].lrValue := STRING_TO_LREAL(sValue);
						END_IF			
				END_IF 
			END_FOR
				byCounterLoop := byCounterLoop + 1;
					byCounterLoop := LIMIT(0,byCounterLoop,250);
						//Back to Step Nr 2
						IF byCounterLoop > byPlaceInArrayInUse THEN iStateCheckValue := 2; EXIT; END_IF 
		END_FOR
		
END_CASE

END_FUNCTION_BLOCK

